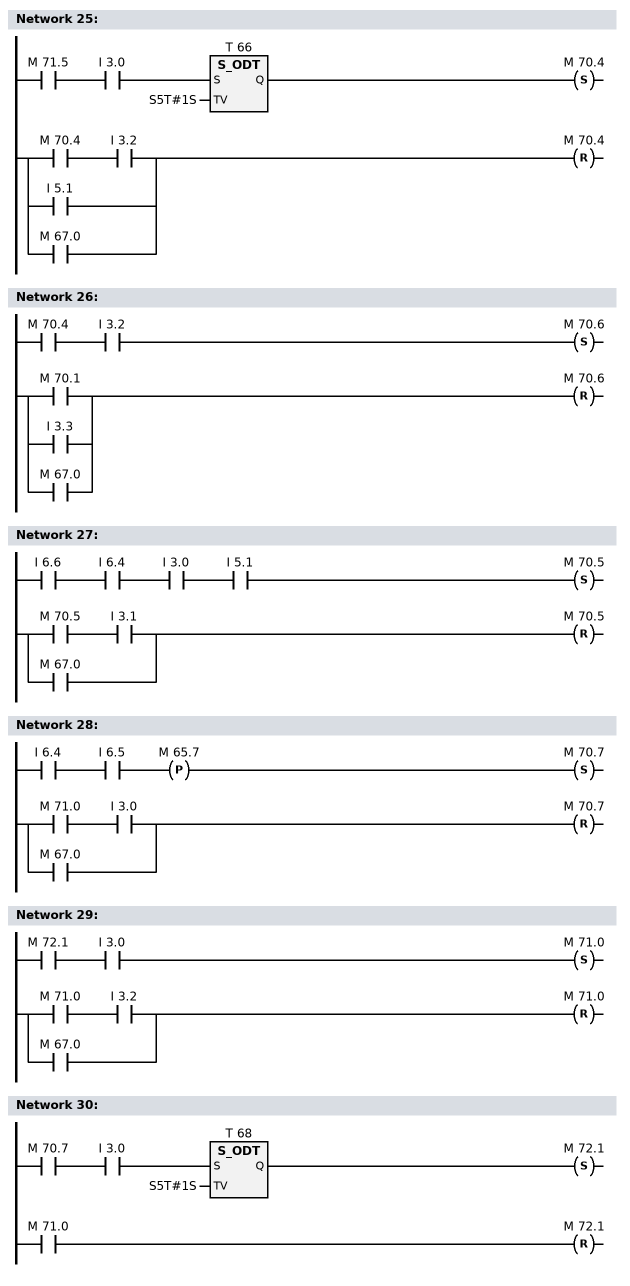
NETWORK
TITLE =
      A(;
      A     M 71.5;
      A     I 3.0;
      L     S5T#1S;
      SD    T 66;
      NOP   0;
      NOP   0;
      NOP   0;
      A     T 66;
      );
      S     M 70.4;
      A(;
      A     M 70.4;
      A     I 3.2;
      O     I 5.1;
      O     M 67.0;
      );
      R     M 70.4;
      NOP   0;
NETWORK
TITLE =
      A     M 70.4;
      A     I 3.2;
      S     M 70.6;
      A(;
      O     M 70.1;
      O     I 3.3;
      O     M 67.0;
      );
      R     M 70.6;
      NOP   0;
NETWORK
TITLE =
      A     I 6.6;
      A     I 6.4;
      A     I 3.0;
      A     I 5.1;
      S     M 70.5;
      A(;
      A     M 70.5;
      A     I 3.1;
      O     M 67.0;
      );
      R     M 70.5;
      NOP   0;
NETWORK
TITLE =
      A     I 6.4;
      A     I 6.5;
      FP    M 65.7;
      S     M 70.7;
      A(;
      A     M 71.0;
      A     I 3.0;
      O     M 67.0;
      );
      R     M 70.7;
      NOP   0;
NETWORK
TITLE =
      A     M 72.1;
      A     I 3.0;
      S     M 71.0;
      A(;
      A     M 71.0;
      A     I 3.2;
      O     M 67.0;
      );
      R     M 71.0;
      NOP   0;
NETWORK
TITLE =
      A(;
      A     M 70.7;
      A     I 3.0;
      L     S5T#1S;
      SD    T 68;
      NOP   0;
      NOP   0;
      NOP   0;
      A     T 68;
      );
      S     M 72.1;
      A     M 71.0;
      R     M 72.1;
      NOP   0;
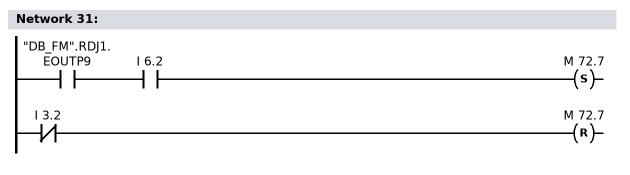
NETWORK
TITLE =
      A     "DB_FM".RDJ1.EOUTP9;
      A     I 6.2;
      S     M 72.7;
      AN    I 3.2;
      R     M 72.7;
      NOP   0;
END_FUNCTION

FUNCTION FC 115 : VOID
VERSION : 0.1
BEGIN
// (block stored without names or comments; labels and parameter names are numbered)
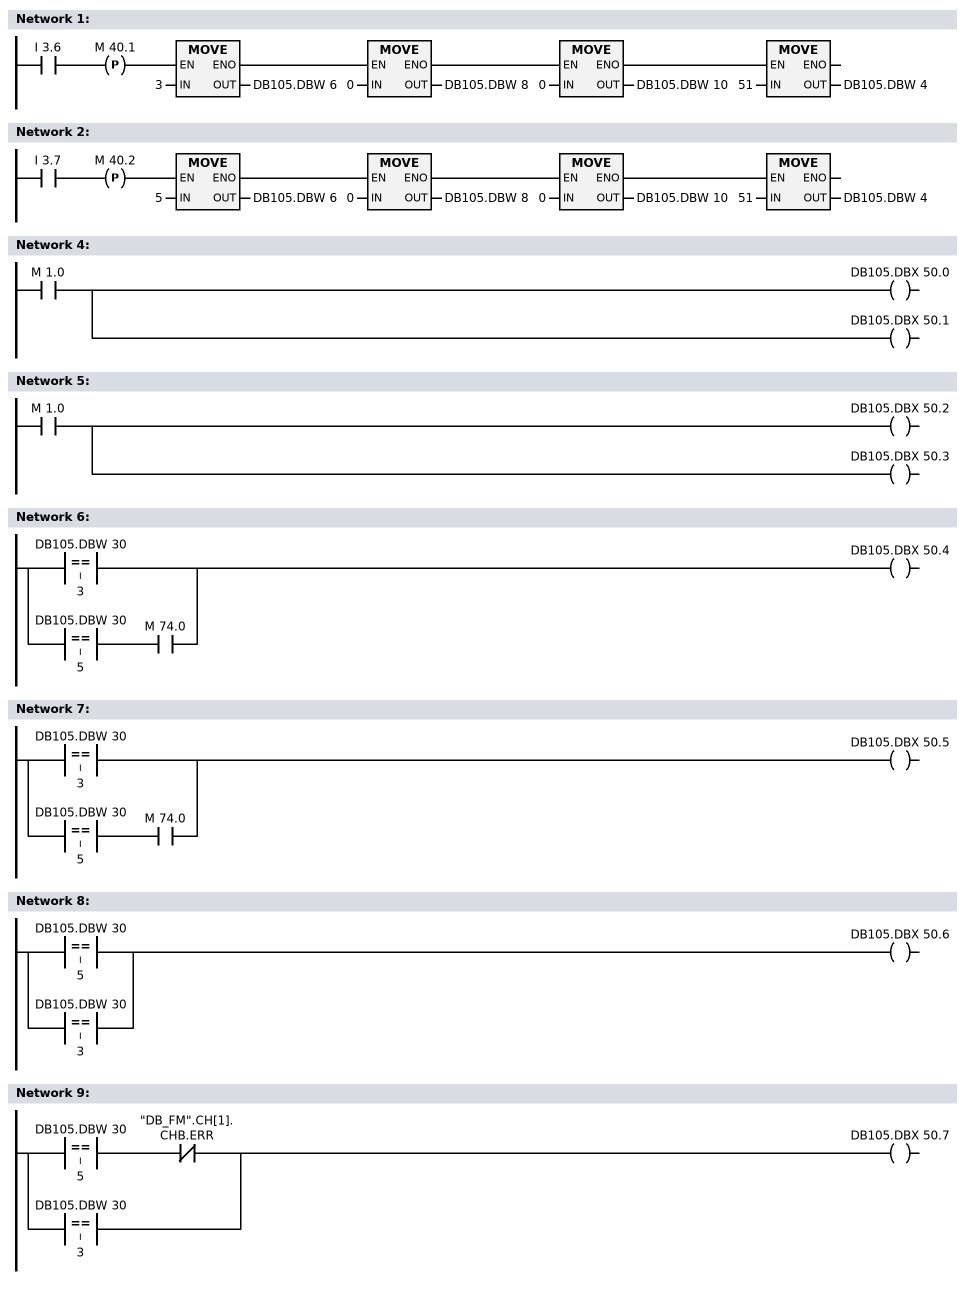
NETWORK
TITLE =
      A(;
      A(;
      A(;
      A     I 3.6;
      FP    M 40.1;
      JNB   M001;
      L     3;
      T     DB105.DBW 6;
      SET;
      SAVE;
      CLR;
M001: A     BR;
      );
      JNB   M002;
      L     0;
      T     DB105.DBW 8;
      SET;
      SAVE;
      CLR;
M002: A     BR;
      );
      JNB   M003;
      L     0;
      T     DB105.DBW 10;
      SET;
      SAVE;
      CLR;
M003: A     BR;
      );
      JNB   M004;
      L     51;
      T     DB105.DBW 4;
M004: NOP   0;
NETWORK
TITLE =
      A(;
      A(;
      A(;
      A     I 3.7;
      FP    M 40.2;
      JNB   M005;
      L     5;
      T     DB105.DBW 6;
      SET;
      SAVE;
      CLR;
M005: A     BR;
      );
      JNB   M006;
      L     0;
      T     DB105.DBW 8;
      SET;
      SAVE;
      CLR;
M006: A     BR;
      );
      JNB   M007;
      L     0;
      T     DB105.DBW 10;
      SET;
      SAVE;
      CLR;
M007: A     BR;
      );
      JNB   M008;
      L     51;
      T     DB105.DBW 4;
M008: NOP   0;
NETWORK
TITLE =
NETWORK
TITLE =
      A     M 1.0;
      =     DB105.DBX 50.0;
      =     DB105.DBX 50.1;
NETWORK
TITLE =
      A     M 1.0;
      =     DB105.DBX 50.2;
      =     DB105.DBX 50.3;
NETWORK
TITLE =
      O(;
      L     DB105.DBW 30;
      L     3;
      ==I;
      );
      O;
      A(;
      L     DB105.DBW 30;
      L     5;
      ==I;
      );
      A     M 74.0;
      =     DB105.DBX 50.4;
NETWORK
TITLE =
      O(;
      L     DB105.DBW 30;
      L     3;
      ==I;
      );
      O;
      A(;
      L     DB105.DBW 30;
      L     5;
      ==I;
      );
      A     M 74.0;
      =     DB105.DBX 50.5;
NETWORK
TITLE =
      O(;
      L     DB105.DBW 30;
      L     5;
      ==I;
      );
      O(;
      L     DB105.DBW 30;
      L     3;
      ==I;
      );
      =     DB105.DBX 50.6;
NETWORK
TITLE =
      A(;
      L     DB105.DBW 30;
      L     5;
      ==I;
      );
      AN    "DB_FM".CH[1].CHB.ERR;
      O(;
      L     DB105.DBW 30;
      L     3;
      ==I;
      );
      =     DB105.DBX 50.7;
END_FUNCTION

FUNCTION FC 118 : VOID
VERSION : 0.1
BEGIN
// (block stored without names or comments; labels and parameter names are numbered)
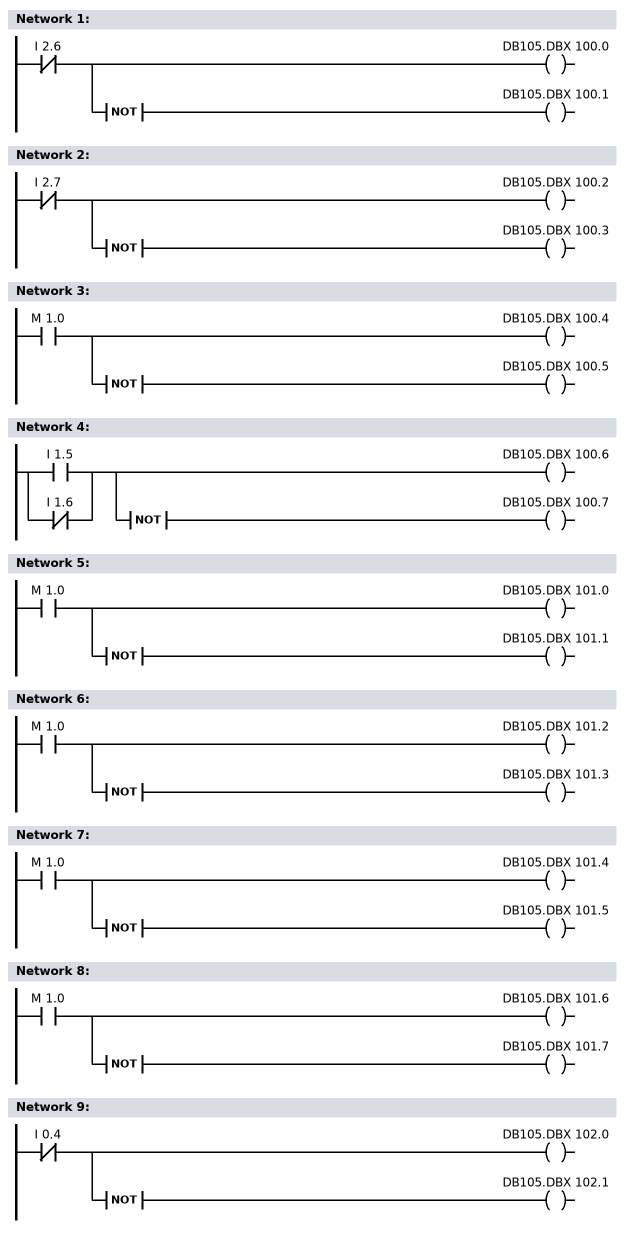
NETWORK
TITLE =
      AN    I 2.6;
      =     L 22.0;
      A     L 22.0;
      BLD   102;
      =     DB105.DBX 100.0;
      A     L 22.0;
      NOT;
      =     DB105.DBX 100.1;
NETWORK
TITLE =
      AN    I 2.7;
      =     L 22.0;
      A     L 22.0;
      BLD   102;
      =     DB105.DBX 100.2;
      A     L 22.0;
      NOT;
      =     DB105.DBX 100.3;
NETWORK
TITLE =
      A     M 1.0;
      =     L 22.0;
      A     L 22.0;
      BLD   102;
      =     DB105.DBX 100.4;
      A     L 22.0;
      NOT;
      =     DB105.DBX 100.5;
NETWORK
TITLE =
      O     I 1.5;
      ON    I 1.6;
      =     L 22.0;
      A     L 22.0;
      BLD   102;
      =     DB105.DBX 100.6;
      A     L 22.0;
      NOT;
      =     DB105.DBX 100.7;
NETWORK
TITLE =
      A     M 1.0;
      =     L 22.0;
      A     L 22.0;
      BLD   102;
      =     DB105.DBX 101.0;
      A     L 22.0;
      NOT;
      =     DB105.DBX 101.1;
NETWORK
TITLE =
      A     M 1.0;
      =     L 22.0;
      A     L 22.0;
      BLD   102;
      =     DB105.DBX 101.2;
      A     L 22.0;
      NOT;
      =     DB105.DBX 101.3;
NETWORK
TITLE =
      A     M 1.0;
      =     L 22.0;
      A     L 22.0;
      BLD   102;
      =     DB105.DBX 101.4;
      A     L 22.0;
      NOT;
      =     DB105.DBX 101.5;
NETWORK
TITLE =
      A     M 1.0;
      =     L 22.0;
      A     L 22.0;
      BLD   102;
      =     DB105.DBX 101.6;
      A     L 22.0;
      NOT;
      =     DB105.DBX 101.7;
NETWORK
TITLE =
      AN    I 0.4;
      =     L 22.0;
      A     L 22.0;
      BLD   102;
      =     DB105.DBX 102.0;
      A     L 22.0;
      NOT;
      =     DB105.DBX 102.1;
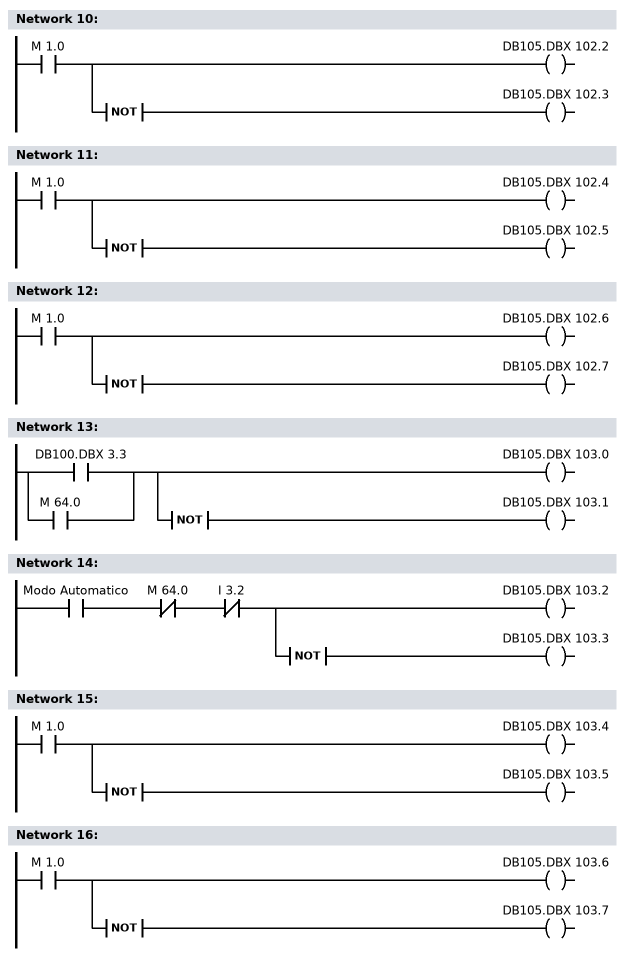
NETWORK
TITLE =
      A     M 1.0;
      =     L 22.0;
      A     L 22.0;
      BLD   102;
      =     DB105.DBX 102.2;
      A     L 22.0;
      NOT;
      =     DB105.DBX 102.3;
NETWORK
TITLE =
      A     M 1.0;
      =     L 22.0;
      A     L 22.0;
      BLD   102;
      =     DB105.DBX 102.4;
      A     L 22.0;
      NOT;
      =     DB105.DBX 102.5;
NETWORK
TITLE =
      A     M 1.0;
      =     L 22.0;
      A     L 22.0;
      BLD   102;
      =     DB105.DBX 102.6;
      A     L 22.0;
      NOT;
      =     DB105.DBX 102.7;
NETWORK
TITLE =
      O     DB100.DBX 3.3;
      O     M 64.0;
      =     L 22.0;
      A     L 22.0;
      BLD   102;
      =     DB105.DBX 103.0;
      A     L 22.0;
      NOT;
      =     DB105.DBX 103.1;
NETWORK
TITLE =
      A     "Modo Automatico";
      AN    M 64.0;
      AN    I 3.2;
      =     L 22.0;
      A     L 22.0;
      BLD   102;
      =     DB105.DBX 103.2;
      A     L 22.0;
      NOT;
      =     DB105.DBX 103.3;
NETWORK
TITLE =
      A     M 1.0;
      =     L 22.0;
      A     L 22.0;
      BLD   102;
      =     DB105.DBX 103.4;
      A     L 22.0;
      NOT;
      =     DB105.DBX 103.5;
NETWORK
TITLE =
      A     M 1.0;
      =     L 22.0;
      A     L 22.0;
      BLD   102;
      =     DB105.DBX 103.6;
      A     L 22.0;
      NOT;
      =     DB105.DBX 103.7;
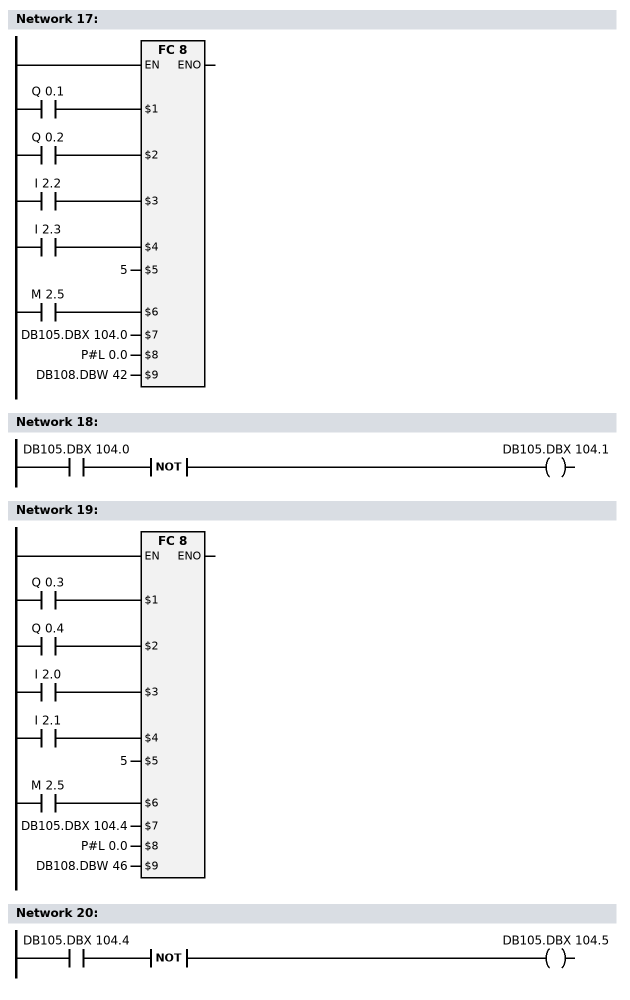
NETWORK
TITLE =
      A     Q 0.1;
      =     L 22.0;
      BLD   103;
      A     Q 0.2;
      =     L 22.1;
      BLD   103;
      A     I 2.2;
      =     L 22.2;
      BLD   103;
      A     I 2.3;
      =     L 22.3;
      BLD   103;
      A     M 2.5;
      =     L 22.4;
      BLD   103;
      CALL  FC 8 (
           $1                       := L 22.0,
           $2                       := L 22.1,
           $3                       := L 22.2,
           $4                       := L 22.3,
           $5                       := 5,
           $6                       := L 22.4,
           $7                       := DB105.DBX 104.0,
           $8                       := P#L 0.0,
           $9                       := DB108.DBW 42);
      NOP   0;
NETWORK
TITLE =
      A     DB105.DBX 104.0;
      NOT;
      =     DB105.DBX 104.1;
NETWORK
TITLE =
      A     Q 0.3;
      =     L 22.0;
      BLD   103;
      A     Q 0.4;
      =     L 22.1;
      BLD   103;
      A     I 2.0;
      =     L 22.2;
      BLD   103;
      A     I 2.1;
      =     L 22.3;
      BLD   103;
      A     M 2.5;
      =     L 22.4;
      BLD   103;
      CALL  FC 8 (
           $1                       := L 22.0,
           $2                       := L 22.1,
           $3                       := L 22.2,
           $4                       := L 22.3,
           $5                       := 5,
           $6                       := L 22.4,
           $7                       := DB105.DBX 104.4,
           $8                       := P#L 0.0,
           $9                       := DB108.DBW 46);
      NOP   0;
NETWORK
TITLE =
      A     DB105.DBX 104.4;
      NOT;
      =     DB105.DBX 104.5;
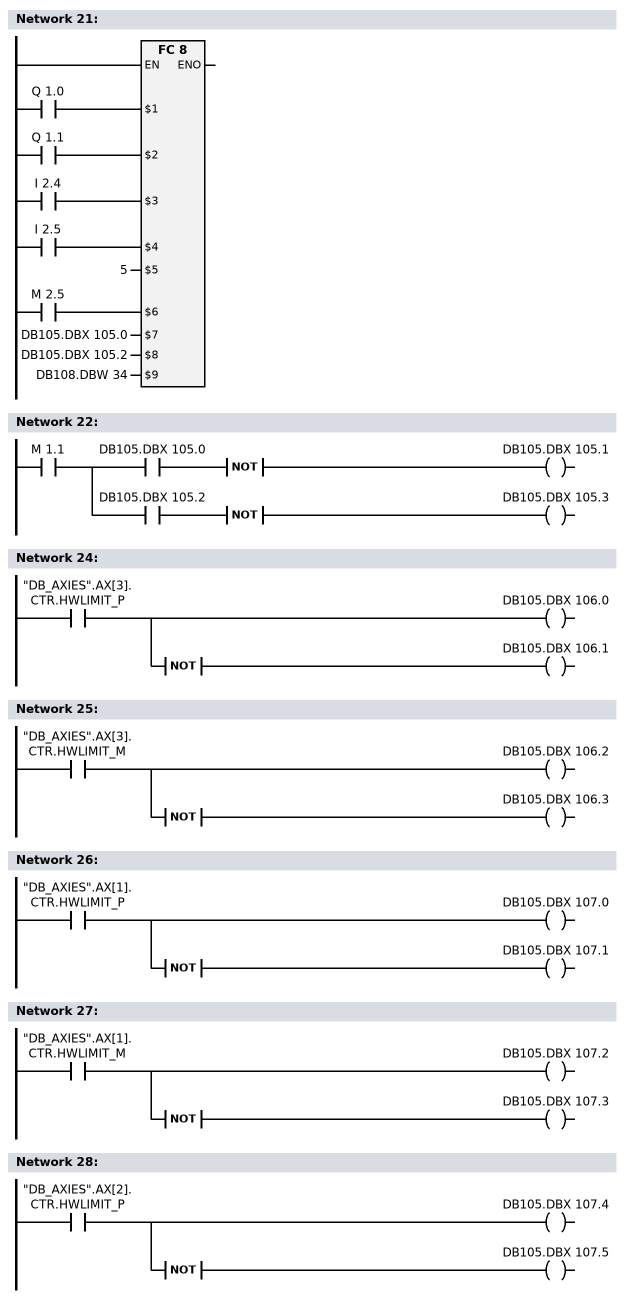
NETWORK
TITLE =
      A     Q 1.0;
      =     L 22.0;
      BLD   103;
      A     Q 1.1;
      =     L 22.1;
      BLD   103;
      A     I 2.4;
      =     L 22.2;
      BLD   103;
      A     I 2.5;
      =     L 22.3;
      BLD   103;
      A     M 2.5;
      =     L 22.4;
      BLD   103;
      CALL  FC 8 (
           $1                       := L 22.0,
           $2                       := L 22.1,
           $3                       := L 22.2,
           $4                       := L 22.3,
           $5                       := 5,
           $6                       := L 22.4,
           $7                       := DB105.DBX 105.0,
           $8                       := DB105.DBX 105.2,
           $9                       := DB108.DBW 34);
      NOP   0;
NETWORK
TITLE =
      A     M 1.1;
      =     L 22.0;
      A     L 22.0;
      A     DB105.DBX 105.0;
      NOT;
      =     DB105.DBX 105.1;
      A     L 22.0;
      A     DB105.DBX 105.2;
      NOT;
      =     DB105.DBX 105.3;
NETWORK
TITLE =
NETWORK
TITLE =
      A     "DB_AXIES".AX[3].CTR.HWLIMIT_P;
      =     L 22.0;
      A     L 22.0;
      BLD   102;
      =     DB105.DBX 106.0;
      A     L 22.0;
      NOT;
      =     DB105.DBX 106.1;
NETWORK
TITLE =
      A     "DB_AXIES".AX[3].CTR.HWLIMIT_M;
      =     L 22.0;
      A     L 22.0;
      BLD   102;
      =     DB105.DBX 106.2;
      A     L 22.0;
      NOT;
      =     DB105.DBX 106.3;
NETWORK
TITLE =
      A     "DB_AXIES".AX[1].CTR.HWLIMIT_P;
      =     L 22.0;
      A     L 22.0;
      BLD   102;
      =     DB105.DBX 107.0;
      A     L 22.0;
      NOT;
      =     DB105.DBX 107.1;
NETWORK
TITLE =
      A     "DB_AXIES".AX[1].CTR.HWLIMIT_M;
      =     L 22.0;
      A     L 22.0;
      BLD   102;
      =     DB105.DBX 107.2;
      A     L 22.0;
      NOT;
      =     DB105.DBX 107.3;
NETWORK
TITLE =
      A     "DB_AXIES".AX[2].CTR.HWLIMIT_P;
      =     L 22.0;
      A     L 22.0;
      BLD   102;
      =     DB105.DBX 107.4;
      A     L 22.0;
      NOT;
      =     DB105.DBX 107.5;
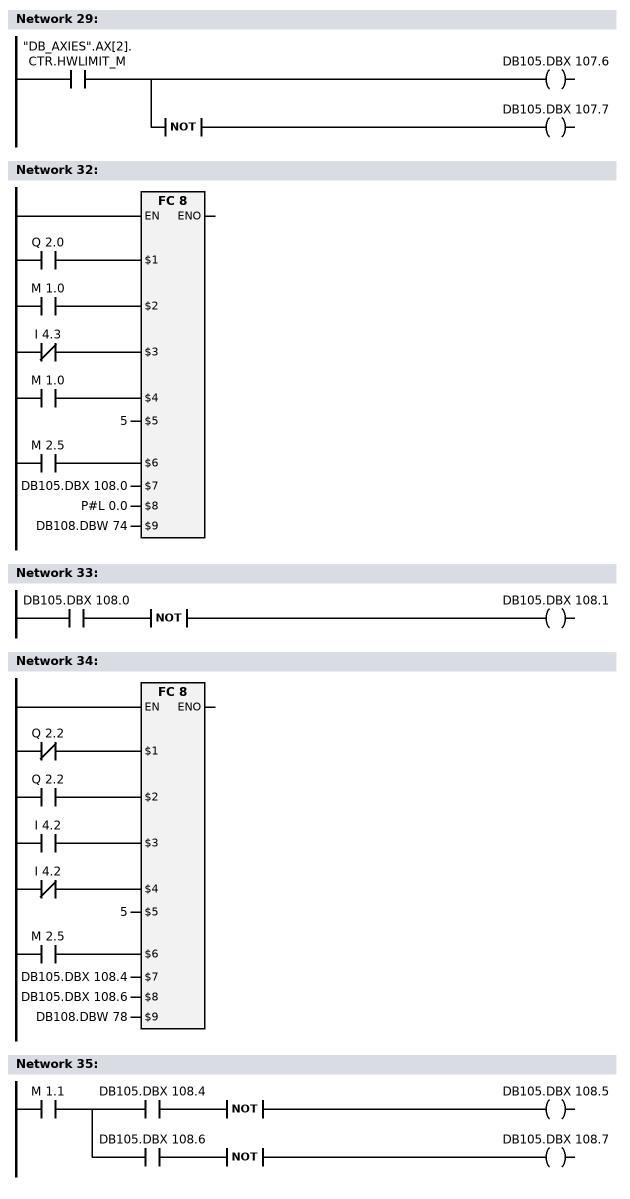
NETWORK
TITLE =
      A     "DB_AXIES".AX[2].CTR.HWLIMIT_M;
      =     L 22.0;
      A     L 22.0;
      BLD   102;
      =     DB105.DBX 107.6;
      A     L 22.0;
      NOT;
      =     DB105.DBX 107.7;
NETWORK
TITLE =
NETWORK
TITLE =
NETWORK
TITLE =
      A     Q 2.0;
      =     L 22.0;
      BLD   103;
      A     M 1.0;
      =     L 22.1;
      BLD   103;
      AN    I 4.3;
      =     L 22.2;
      BLD   103;
      A     M 1.0;
      =     L 22.3;
      BLD   103;
      A     M 2.5;
      =     L 22.4;
      BLD   103;
      CALL  FC 8 (
           $1                       := L 22.0,
           $2                       := L 22.1,
           $3                       := L 22.2,
           $4                       := L 22.3,
           $5                       := 5,
           $6                       := L 22.4,
           $7                       := DB105.DBX 108.0,
           $8                       := P#L 0.0,
           $9                       := DB108.DBW 74);
      NOP   0;
NETWORK
TITLE =
      A     DB105.DBX 108.0;
      NOT;
      =     DB105.DBX 108.1;
NETWORK
TITLE =
      AN    Q 2.2;
      =     L 22.0;
      BLD   103;
      A     Q 2.2;
      =     L 22.1;
      BLD   103;
      A     I 4.2;
      =     L 22.2;
      BLD   103;
      AN    I 4.2;
      =     L 22.3;
      BLD   103;
      A     M 2.5;
      =     L 22.4;
      BLD   103;
      CALL  FC 8 (
           $1                       := L 22.0,
           $2                       := L 22.1,
           $3                       := L 22.2,
           $4                       := L 22.3,
           $5                       := 5,
           $6                       := L 22.4,
           $7                       := DB105.DBX 108.4,
           $8                       := DB105.DBX 108.6,
           $9                       := DB108.DBW 78);
      NOP   0;
NETWORK
TITLE =
      A     M 1.1;
      =     L 22.0;
      A     L 22.0;
      A     DB105.DBX 108.4;
      NOT;
      =     DB105.DBX 108.5;
      A     L 22.0;
      A     DB105.DBX 108.6;
      NOT;
      =     DB105.DBX 108.7;
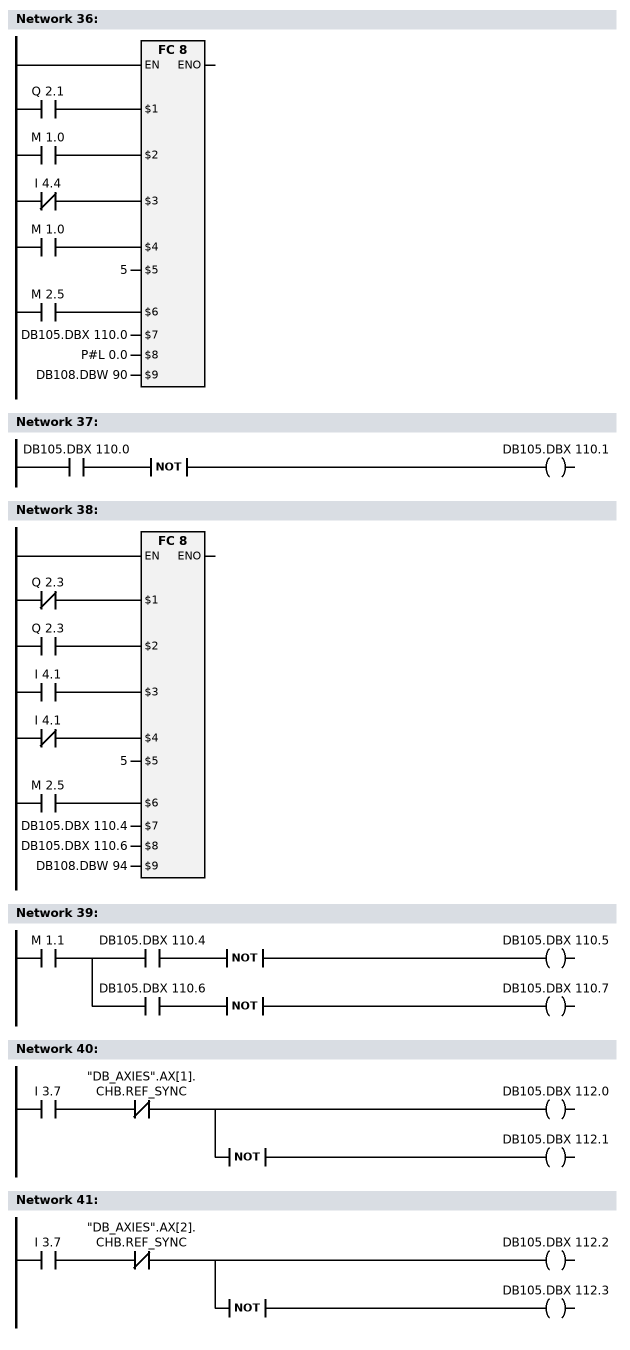
NETWORK
TITLE =
      A     Q 2.1;
      =     L 22.0;
      BLD   103;
      A     M 1.0;
      =     L 22.1;
      BLD   103;
      AN    I 4.4;
      =     L 22.2;
      BLD   103;
      A     M 1.0;
      =     L 22.3;
      BLD   103;
      A     M 2.5;
      =     L 22.4;
      BLD   103;
      CALL  FC 8 (
           $1                       := L 22.0,
           $2                       := L 22.1,
           $3                       := L 22.2,
           $4                       := L 22.3,
           $5                       := 5,
           $6                       := L 22.4,
           $7                       := DB105.DBX 110.0,
           $8                       := P#L 0.0,
           $9                       := DB108.DBW 90);
      NOP   0;
NETWORK
TITLE =
      A     DB105.DBX 110.0;
      NOT;
      =     DB105.DBX 110.1;
NETWORK
TITLE =
      AN    Q 2.3;
      =     L 22.0;
      BLD   103;
      A     Q 2.3;
      =     L 22.1;
      BLD   103;
      A     I 4.1;
      =     L 22.2;
      BLD   103;
      AN    I 4.1;
      =     L 22.3;
      BLD   103;
      A     M 2.5;
      =     L 22.4;
      BLD   103;
      CALL  FC 8 (
           $1                       := L 22.0,
           $2                       := L 22.1,
           $3                       := L 22.2,
           $4                       := L 22.3,
           $5                       := 5,
           $6                       := L 22.4,
           $7                       := DB105.DBX 110.4,
           $8                       := DB105.DBX 110.6,
           $9                       := DB108.DBW 94);
      NOP   0;
NETWORK
TITLE =
      A     M 1.1;
      =     L 22.0;
      A     L 22.0;
      A     DB105.DBX 110.4;
      NOT;
      =     DB105.DBX 110.5;
      A     L 22.0;
      A     DB105.DBX 110.6;
      NOT;
      =     DB105.DBX 110.7;
NETWORK
TITLE =
      A     I 3.7;
      AN    "DB_AXIES".AX[1].CHB.REF_SYNC;
      =     L 22.0;
      A     L 22.0;
      BLD   102;
      =     DB105.DBX 112.0;
      A     L 22.0;
      NOT;
      =     DB105.DBX 112.1;
NETWORK
TITLE =
      A     I 3.7;
      AN    "DB_AXIES".AX[2].CHB.REF_SYNC;
      =     L 22.0;
      A     L 22.0;
      BLD   102;
      =     DB105.DBX 112.2;
      A     L 22.0;
      NOT;
      =     DB105.DBX 112.3;
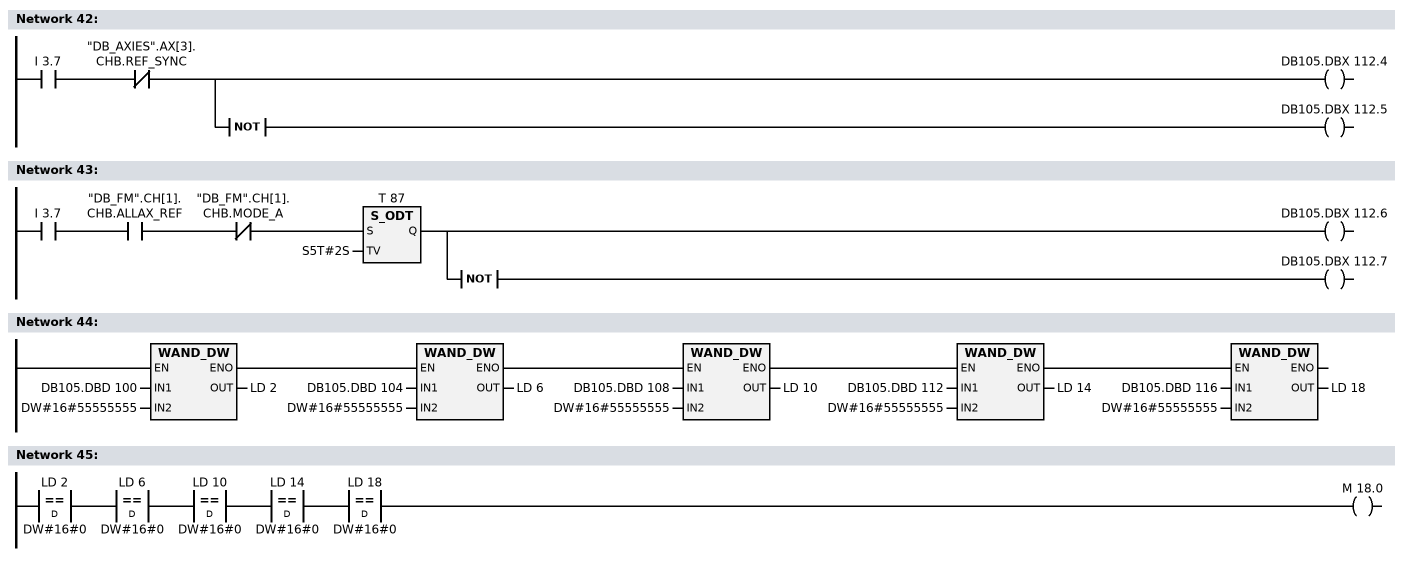
NETWORK
TITLE =
      A     I 3.7;
      AN    "DB_AXIES".AX[3].CHB.REF_SYNC;
      =     L 22.0;
      A     L 22.0;
      BLD   102;
      =     DB105.DBX 112.4;
      A     L 22.0;
      NOT;
      =     DB105.DBX 112.5;
NETWORK
TITLE =
      A     I 3.7;
      A     "DB_FM".CH[1].CHB.ALLAX_REF;
      AN    "DB_FM".CH[1].CHB.MODE_A;
      L     S5T#2S;
      SD    T 87;
      NOP   0;
      NOP   0;
      NOP   0;
      A     T 87;
      =     L 22.0;
      A     L 22.0;
      BLD   102;
      =     DB105.DBX 112.6;
      A     L 22.0;
      NOT;
      =     DB105.DBX 112.7;
NETWORK
TITLE =
      A(;
      A(;
      A(;
      A(;
      L     DB105.DBD 100;
      L     DW#16#55555555;
      AD;
      T     LD 2;
      SET;
      SAVE;
      CLR;
      A     BR;
      );
      JNB   M001;
      L     DB105.DBD 104;
      L     DW#16#55555555;
      AD;
      T     LD 6;
      SET;
      SAVE;
      CLR;
M001: A     BR;
      );
      JNB   M002;
      L     DB105.DBD 108;
      L     DW#16#55555555;
      AD;
      T     LD 10;
      SET;
      SAVE;
      CLR;
M002: A     BR;
      );
      JNB   M003;
      L     DB105.DBD 112;
      L     DW#16#55555555;
      AD;
      T     LD 14;
      SET;
      SAVE;
      CLR;
M003: A     BR;
      );
      JNB   M004;
      L     DB105.DBD 116;
      L     DW#16#55555555;
      AD;
      T     LD 18;
M004: NOP   0;
NETWORK
TITLE =
      A(;
      L     LD 2;
      L     DW#16#0;
      ==D;
      );
      A(;
      L     LD 6;
      L     DW#16#0;
      ==D;
      );
      A(;
      L     LD 10;
      L     DW#16#0;
      ==D;
      );
      A(;
      L     LD 14;
      L     DW#16#0;
      ==D;
      );
      A(;
      L     LD 18;
      L     DW#16#0;
      ==D;
      );
      =     M 18.0;
END_FUNCTION

FUNCTION FC 119 : VOID
VERSION : 0.1
BEGIN
// (block stored without names or comments; labels and parameter names are numbered)
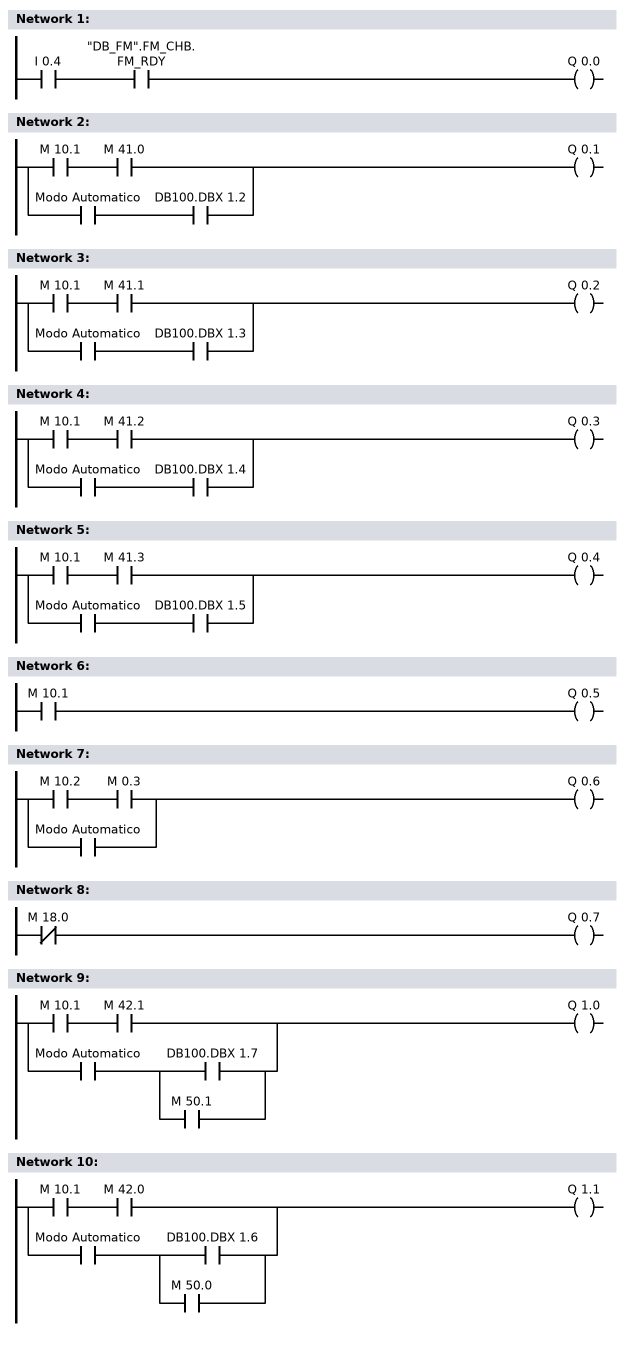
NETWORK
TITLE =
      A     I 0.4;
      A     "DB_FM".FM_CHB.FM_RDY;
      =     Q 0.0;
NETWORK
TITLE =
      A     M 10.1;
      A     M 41.0;
      O;
      A     "Modo Automatico";
      A     DB100.DBX 1.2;
      =     Q 0.1;
NETWORK
TITLE =
      A     M 10.1;
      A     M 41.1;
      O;
      A     "Modo Automatico";
      A     DB100.DBX 1.3;
      =     Q 0.2;
NETWORK
TITLE =
      A     M 10.1;
      A     M 41.2;
      O;
      A     "Modo Automatico";
      A     DB100.DBX 1.4;
      =     Q 0.3;
NETWORK
TITLE =
      A     M 10.1;
      A     M 41.3;
      O;
      A     "Modo Automatico";
      A     DB100.DBX 1.5;
      =     Q 0.4;
NETWORK
TITLE =
      A     M 10.1;
      =     Q 0.5;
NETWORK
TITLE =
      A     M 10.2;
      A     M 0.3;
      O     "Modo Automatico";
      =     Q 0.6;
NETWORK
TITLE =
      AN    M 18.0;
      =     Q 0.7;
NETWORK
TITLE =
      A     M 10.1;
      A     M 42.1;
      O;
      A     "Modo Automatico";
      A(;
      O     DB100.DBX 1.7;
      O     M 50.1;
      );
      =     Q 1.0;
NETWORK
TITLE =
      A     M 10.1;
      A     M 42.0;
      O;
      A     "Modo Automatico";
      A(;
      O     DB100.DBX 1.6;
      O     M 50.0;
      );
      =     Q 1.1;
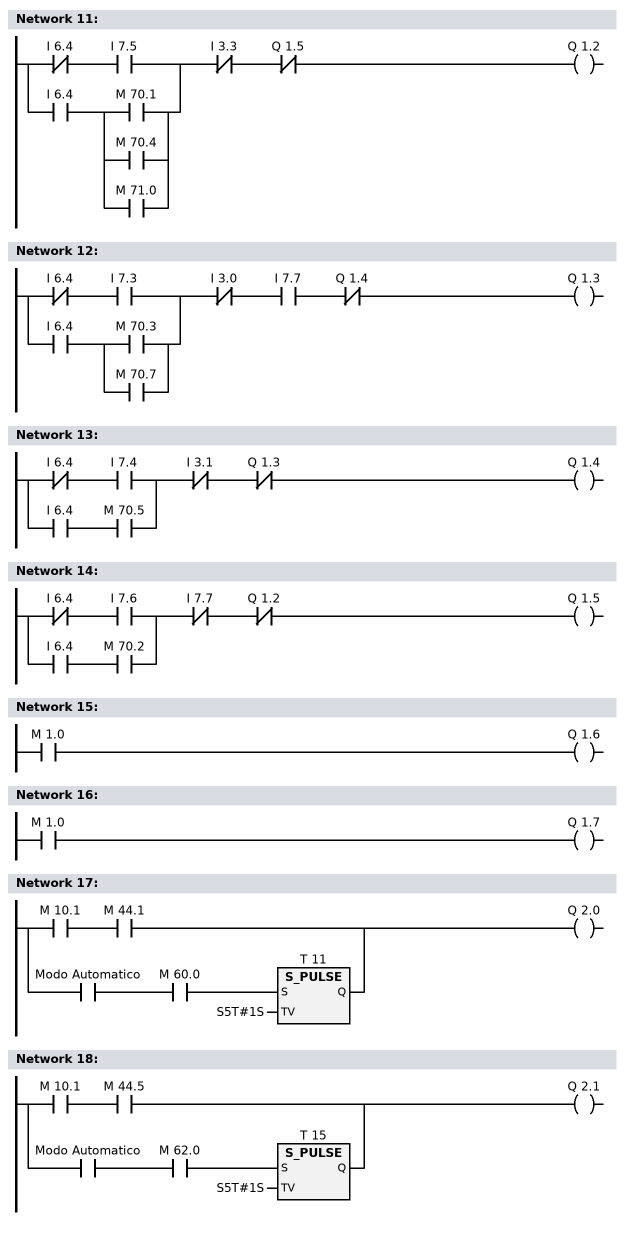
NETWORK
TITLE =
      A(;
      AN    I 6.4;
      A     I 7.5;
      O;
      A     I 6.4;
      A(;
      O     M 70.1;
      O     M 70.4;
      O     M 71.0;
      );
      );
      AN    I 3.3;
      AN    Q 1.5;
      =     Q 1.2;
NETWORK
TITLE =
      A(;
      AN    I 6.4;
      A     I 7.3;
      O;
      A     I 6.4;
      A(;
      O     M 70.3;
      O     M 70.7;
      );
      );
      AN    I 3.0;
      A     I 7.7;
      AN    Q 1.4;
      =     Q 1.3;
NETWORK
TITLE =
      A(;
      AN    I 6.4;
      A     I 7.4;
      O;
      A     I 6.4;
      A     M 70.5;
      );
      AN    I 3.1;
      AN    Q 1.3;
      =     Q 1.4;
NETWORK
TITLE =
      A(;
      AN    I 6.4;
      A     I 7.6;
      O;
      A     I 6.4;
      A     M 70.2;
      );
      AN    I 7.7;
      AN    Q 1.2;
      =     Q 1.5;
NETWORK
TITLE =
      A     M 1.0;
      =     Q 1.6;
NETWORK
TITLE =
      A     M 1.0;
      =     Q 1.7;
NETWORK
TITLE =
      A     M 10.1;
      A     M 44.1;
      O(;
      A     "Modo Automatico";
      A     M 60.0;
      L     S5T#1S;
      SP    T 11;
      NOP   0;
      NOP   0;
      NOP   0;
      A     T 11;
      );
      =     Q 2.0;
NETWORK
TITLE =
      A     M 10.1;
      A     M 44.5;
      O(;
      A     "Modo Automatico";
      A     M 62.0;
      L     S5T#1S;
      SP    T 15;
      NOP   0;
      NOP   0;
      NOP   0;
      A     T 15;
      );
      =     Q 2.1;
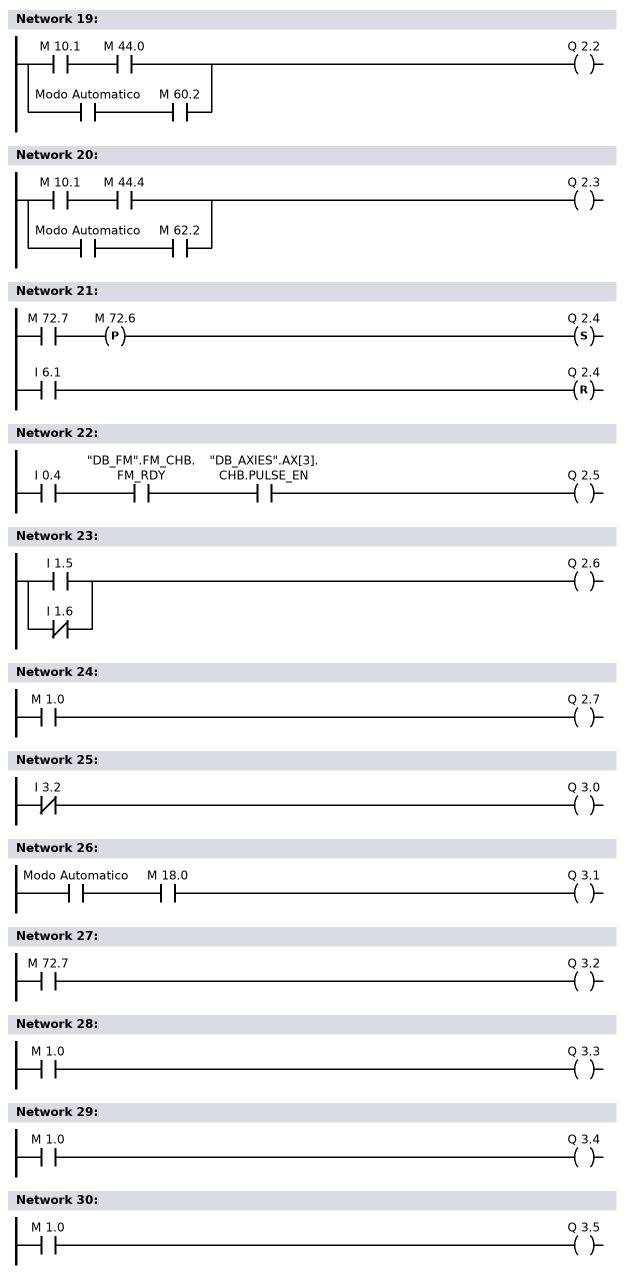
NETWORK
TITLE =
      A     M 10.1;
      A     M 44.0;
      O;
      A     "Modo Automatico";
      A     M 60.2;
      =     Q 2.2;
NETWORK
TITLE =
      A     M 10.1;
      A     M 44.4;
      O;
      A     "Modo Automatico";
      A     M 62.2;
      =     Q 2.3;
NETWORK
TITLE =
      A     M 72.7;
      FP    M 72.6;
      S     Q 2.4;
      A     I 6.1;
      R     Q 2.4;
      NOP   0;
NETWORK
TITLE =
      A     I 0.4;
      A     "DB_FM".FM_CHB.FM_RDY;
      A     "DB_AXIES".AX[3].CHB.PULSE_EN;
      =     Q 2.5;
NETWORK
TITLE =
      O     I 1.5;
      ON    I 1.6;
      =     Q 2.6;
NETWORK
TITLE =
      A     M 1.0;
      =     Q 2.7;
NETWORK
TITLE =
      AN    I 3.2;
      =     Q 3.0;
NETWORK
TITLE =
      A     "Modo Automatico";
      A     M 18.0;
      =     Q 3.1;
NETWORK
TITLE =
      A     M 72.7;
      =     Q 3.2;
NETWORK
TITLE =
      A     M 1.0;
      =     Q 3.3;
NETWORK
TITLE =
      A     M 1.0;
      =     Q 3.4;
NETWORK
TITLE =
      A     M 1.0;
      =     Q 3.5;
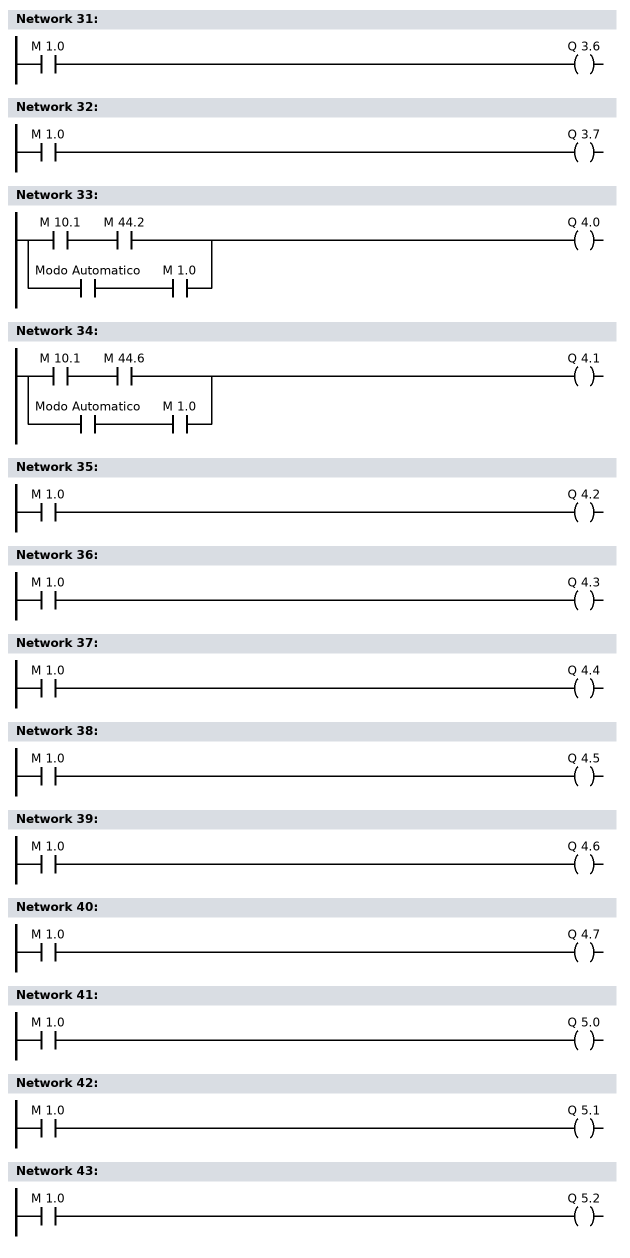
NETWORK
TITLE =
      A     M 1.0;
      =     Q 3.6;
NETWORK
TITLE =
      A     M 1.0;
      =     Q 3.7;
NETWORK
TITLE =
      A     M 10.1;
      A     M 44.2;
      O;
      A     "Modo Automatico";
      A     M 1.0;
      =     Q 4.0;
NETWORK
TITLE =
      A     M 10.1;
      A     M 44.6;
      O;
      A     "Modo Automatico";
      A     M 1.0;
      =     Q 4.1;
NETWORK
TITLE =
      A     M 1.0;
      =     Q 4.2;
NETWORK
TITLE =
      A     M 1.0;
      =     Q 4.3;
NETWORK
TITLE =
      A     M 1.0;
      =     Q 4.4;
NETWORK
TITLE =
      A     M 1.0;
      =     Q 4.5;
NETWORK
TITLE =
      A     M 1.0;
      =     Q 4.6;
NETWORK
TITLE =
      A     M 1.0;
      =     Q 4.7;
NETWORK
TITLE =
      A     M 1.0;
      =     Q 5.0;
NETWORK
TITLE =
      A     M 1.0;
      =     Q 5.1;
NETWORK
TITLE =
      A     M 1.0;
      =     Q 5.2;
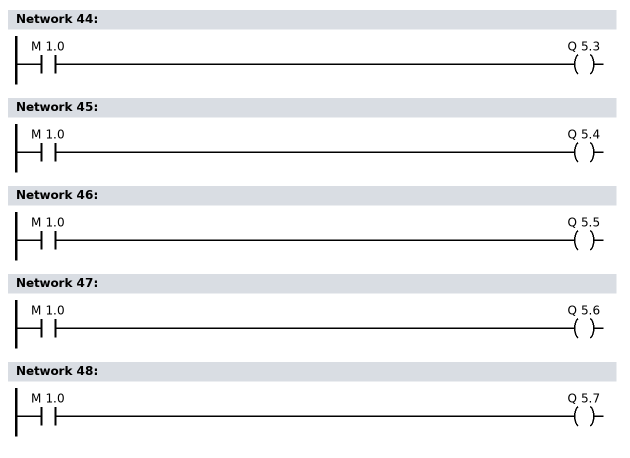
NETWORK
TITLE =
      A     M 1.0;
      =     Q 5.3;
NETWORK
TITLE =
      A     M 1.0;
      =     Q 5.4;
NETWORK
TITLE =
      A     M 1.0;
      =     Q 5.5;
NETWORK
TITLE =
      A     M 1.0;
      =     Q 5.6;
NETWORK
TITLE =
      A     M 1.0;
      =     Q 5.7;
END_FUNCTION

DATA_BLOCK DB 2
VERSION : 0.0
BEGIN
// 66 bytes; values not shown
END_DATA_BLOCK

// DB 7: know-how protected block, not included

DATA_BLOCK DB 15
AUTHOR : AuD_MCE8
FAMILY : FM357_2
NAME : BF_DB15
VERSION : 2.1
FB 6
BEGIN
END_DATA_BLOCK

// DB 16: know-how protected block, not included

// DB 17: know-how protected block, not included

// DB 19: know-how protected block, not included

// DB 20: know-how protected block, not included

DATA_BLOCK "DB_FM"	// DB 30
VERSION : 0.1
  STRUCT
   MOD_ADDR : INT ;	// Module address
   CH_NO : BYTE ;	// No. of channels
   AX_NO : BYTE ;	// No. of axes
   BF_ERR : WORD ;	// Basic function error
   WRJOB1 : BOOL ;	// Write request 1
   WRJOB2 : BOOL ;	// Write request 2
   BIT6_2 : BOOL ;	// Reserved
   BIT6_3 : BOOL ;	// Reserved
   BIT6_4 : BOOL ;	// Reserved
   BIT6_5 : BOOL ;	// Reserved
   BIT6_6 : BOOL ;	// Reserved
   BIT6_7 : BOOL ;	// Reserved
   ERR_WRJOB1 : BOOL ;	// Error in write request 1
   ERR_WRJOB2 : BOOL ;	// Error in write request 2
   BIT7_2 : BOOL ;	// Reserved
   BIT7_3 : BOOL ;	// Reserved
   BIT7_4 : BOOL ;	// Reserved
   BIT7_5 : BOOL ;	// Reserved
   BIT7_6 : BOOL ;	// Reserved
   BIT7_7 : BOOL ;	// Reserved
   RDJOB1 : BOOL ;	// Read request 1
   RDJOB2 : BOOL ;	// Read request 2
   BIT8_2 : BOOL ;	// Reserved
   BIT8_3 : BOOL ;	// Reserved
   BIT8_4 : BOOL ;	// Reserved
   BIT8_5 : BOOL ;	// Reserved
   BIT8_6 : BOOL ;	// Reserved
   BIT8_7 : BOOL ;	// Reserved
   ERR_RDJOB1 : BOOL ;	// Error in read request 1
   ERR_RDJOB2 : BOOL ;	// Error in read request 2
   BIT9_2 : BOOL ;	// Reserved
   BIT9_3 : BOOL ;	// Reserved
   BIT9_4 : BOOL ;	// Reserved
   BIT9_5 : BOOL ;	// Reserved
   BIT9_6 : BOOL ;	// Reserved
   BIT9_7 : BOOL ;	// Reserved
   CONNECT : BOOL ;	// Readiness to communicate
   RESTART : BOOL ;	// FM Restart
   STARTUP : BOOL ;	// FM Startup
   BIT10_3 : BOOL ;	// Reserved
   BIT10_4 : BOOL ;	// Reserved
   BIT10_5 : BOOL ;	// Reserved
   BIT10_6 : BOOL ;	// Reserved
   BIT10_7 : BOOL ;	// Reserved
   PRES_TEST : BOOL ;	// Start-up window: Request for TEST mode
   ACT_TEST : BOOL ;	// User: Enable TEST mode
   BIT11_2 : BOOL ;	// Reserved
   BIT11_3 : BOOL ;	// Reserved
   BIT11_4 : BOOL ;	// Reserved
   BIT11_5 : BOOL ;	// Reserved
   BIT11_6 : BOOL ;	// Reserved
   BIT11_7 : BOOL ;	// Reserved
   BYTE12_19 : ARRAY  [1 .. 8 ] OF BYTE ;	// Reserved
   FM_CTR : STRUCT 	// FM CONTROL SIGNALS
    BIT0_0 : BOOL ;	// Reserved
    EM_STOP : BOOL ;	// EMERGENCY STOP
    ACKN_EM_STOP : BOOL ;	// EMERGENCY STOP acknowledgement
    BIT0_3 : BOOL ;	// Reserved
    BIT0_4 : BOOL ;	// Reserved
    BIT0_5 : BOOL ;	// Reserved
    BIT0_6 : BOOL ;	// Reserved
    BIT0_7 : BOOL ;	// Reserved
    BIT1_0 : BOOL ;	// Reserved
    ACT_POS : BOOL ;	// Request actual values
    DIS_TOGO : BOOL ;	// Request distances to go
    BIT1_3 : BOOL ;	// Reserved
    BIT1_4 : BOOL ;	// Reserved
    BIT1_5 : BOOL ;	// Reserved
    BIT1_6 : BOOL ;	// Reserved
    BIT1_7 : BOOL ;	// Reserved
    CPU_VAR : WORD ;	// CPU variables(write)
    BYTE4_9 : ARRAY  [1 .. 6 ] OF BYTE ;	// Reserved
   END_STRUCT ;
   FM_CHB : STRUCT 	// FM CHECKBACK SIGNALS
    PROBE1 : BOOL ;	// Probe 1 actuated
    PROBE2 : BOOL ;	// Probe 2 actuated
    BIT0_2 : BOOL ;	// Reserved
    BIT0_3 : BOOL ;	// Reserved
    BIT0_4 : BOOL ;	// Reserved
    BIT0_5 : BOOL ;	// Reserved
    BIT0_6 : BOOL ;	// Reserved
    FM_RDY : BOOL ;	// FM ready
    FM_ERR : BOOL ;	// FM error is active
    EM_STOP : BOOL ;	// EMERGENCY STOP active
    BIT1_2 : BOOL ;	// Reserved
    BIT1_3 : BOOL ;	// Reserved
    BIT1_4 : BOOL ;	// Reserved
    BIT1_5 : BOOL ;	// Reserved
    BIT1_6 : BOOL ;	// Reserved
    BATT_ERR : BOOL ;	// FM battery fault
    SWCAM_M1 : BOOL ;	// Software cam MINUS 1
    SWCAM_M2 : BOOL ;	// Software cam MINUS 2
    SWCAM_M3 : BOOL ;	// Software cam MINUS 3
    SWCAM_M4 : BOOL ;	// Software cam MINUS 4
    SWCAM_M5 : BOOL ;	// Software cam MINUS 5
    SWCAM_M6 : BOOL ;	// Software cam MINUS 6
    SWCAM_M7 : BOOL ;	// Software cam MINUS 7
    SWCAM_M8 : BOOL ;	// Software cam MINUS 8
    SWCAM_P1 : BOOL ;	// Software cam PLUS 1
    SWCAM_P2 : BOOL ;	// Software cam PLUS 2
    SWCAM_P3 : BOOL ;	// Software cam PLUS 3
    SWCAM_P4 : BOOL ;	// Software cam PLUS 4
    SWCAM_P5 : BOOL ;	// Software cam PLUS 5
    SWCAM_P6 : BOOL ;	// Software cam PLUS 6
    SWCAM_P7 : BOOL ;	// Software cam PLUS 7
    SWCAM_P8 : BOOL ;	// Software cam PLUS 8
    CPU_VAR : WORD ;	// CPU variables (read)
    BYTE6_9 : ARRAY  [1 .. 4 ] OF BYTE ;	// Reserved
   END_STRUCT ;
   BYTE40_99 : ARRAY  [1 .. 60 ] OF BYTE ;	// Reserved
   CH : ARRAY  [1 .. 4 ] OF STRUCT 	// CHANNEL SIGNALS
    CTR : STRUCT 	// CHANNEL CONTROL SIGNALS
     MODE_A : BOOL ;	// Automatic mode
     MODE_MDI : BOOL ;	// MDI block mode (FM357-H)
     MODE_JOG : BOOL ;	// Jog mode
     BIT0_3 : BOOL ;	// Reserved
     BIT0_4 : BOOL ;	// Reserved
     BIT0_5 : BOOL ;	// Reserved
     BIT0_6 : BOOL ;	// Reserved
     BIT0_7 : BOOL ;	// Reserved
     TEACH_IN : BOOL ;	// Teach-In (FM357-H)
     REPOS : BOOL ;	// Repositioning (FM357-H)
     REF_POINT : BOOL ;	// Reference point approach
     BIT1_3 : BOOL ;	// Reserved
     BIT1_4 : BOOL ;	// Reserved
     BIT1_5 : BOOL ;	// Reserved
     BIT1_6 : BOOL ;	// Reserved
     BIT1_7 : BOOL ;	// Reserved
     INC1 : BOOL ;	// Increment size 1 increment
     INC10 : BOOL ;	// Increment size 10 increments
     INC100 : BOOL ;	// Increment size 100 increments
     INC1000 : BOOL ;	// Increment size 1000 increments
     INC10000 : BOOL ;	// Increment size 10000 increments
     INC_VAR : BOOL ;	// Increment variable (FM357-H)
     CONT_TRAV : BOOL ;	// Continuous traverse
     BIT2_7 : BOOL ;	// Reserved
     BIT3_0 : BOOL ;	// Reserved
     BIT3_1 : BOOL ;	// Reserved
     BIT3_2 : BOOL ;	// Reserved
     BIT3_3 : BOOL ;	// Reserved
     SGL_BL : BOOL ;	// Activate single block
     M1 : BOOL ;	// Activate M1
     DRUN_FD : BOOL ;	// Dry run feed (FM357-H)
     BIT3_7 : BOOL ;	// Reserved
     BIT4_0 : BOOL ;	// Reserved
     BIT4_1 : BOOL ;	// Reserved
     BIT4_2 : BOOL ;	// Reserved
     BIT4_3 : BOOL ;	// Reserved
     BIT4_4 : BOOL ;	// Reserved
     BIT4_5 : BOOL ;	// Reserved
     BIT4_6 : BOOL ;	// Reserved
     PROG_TEST : BOOL ;	// Activate program test (FM357-H)
     SKIP_BL : BOOL ;	// Activate skip block
     BIT5_1 : BOOL ;	// Reserved
     BIT5_2 : BOOL ;	// Reserved
     BIT5_3 : BOOL ;	// Reserved
     BIT5_4 : BOOL ;	// Reserved
     BIT5_5 : BOOL ;	// Reserved
     BIT5_6 : BOOL ;	// Reserved
     BIT5_7 : BOOL ;	// Reserved
     FD_OVERR : BYTE ;	// Path override
     FD_DISA : BOOL ;	// Activate feed disable
     RDIN_DISA : BOOL ;	// Read-in disable
     DELDIS_TOGO : BOOL ;	// Delete distance to go
     BIT7_3 : BOOL ;	// Reserved
     BIT7_4 : BOOL ;	// Reserved
     BIT7_5 : BOOL ;	// Reserved
     FD_OVERR_RTR : BOOL ;	// Path override rapid traverse operative
     FD_OVERR_FDR : BOOL ;	// Path override feedrate operative
     START_DISA : BOOL ;	// Activate start disable
     START : BOOL ;	// Start
     STOP_BL : BOOL ;	// Activate stop at block limit
     STOP : BOOL ;	// Stop
     BIT8_4 : BOOL ;	// Reserved
     BIT8_5 : BOOL ;	// Reserved
     BIT8_6 : BOOL ;	// Reserved
     RESET : BOOL ;	// Reset
     ACKN_AUXILF : BOOL ;	// Acknowledge aux. function
     BIT9_1 : BOOL ;	// Reserved
     BIT9_2 : BOOL ;	// Reserved
     BIT9_3 : BOOL ;	// Reserved
     BIT9_4 : BOOL ;	// Reserved
     BIT9_5 : BOOL ;	// Reserved
     BIT9_6 : BOOL ;	// Reserved
     BIT9_7 : BOOL ;	// Reserved
     BIT10_0 : BOOL ;	// Reserved
     BIT10_1 : BOOL ;	// Reserved
     BIT10_2 : BOOL ;	// Reserved
     BIT10_3 : BOOL ;	// Reserved
     BIT10_4 : BOOL ;	// Reserved
     BIT10_5 : BOOL ;	// Reserved
     BIT10_6 : BOOL ;	// Reserved
     START_ASUP : BOOL ;	// Start "Asynchronous subroutine"
     BYTE11 : BYTE ;	// Reserved
     WORD12 : WORD ;	// Reserved
     BIT14_0 : BOOL ;	// Reserved
     BIT14_1 : BOOL ;	// Reserved
     BIT14_2 : BOOL ;	// Reserved
     FD_STOP_GEOA1 : BOOL ;	// Feed stop geometry axis 1 (FM357-H)
     TR_DISA_GEOA1 : BOOL ;	// Traverse disable geometry axis 1 (FM357-H)
     RTR_OVERL_GEOA1 : BOOL ;	// Rapid traverse override geometry axis 1 (FM357-H)
     DIR_M_GEOA1 : BOOL ;	// MINUS direction geometry axis  1(FM357-H)
     DIR_P_GEOA1 : BOOL ;	// PLUS direction geometry axis 1 (FM357-H)
     BIT15_0 : BOOL ;	// Reserved
     BIT15_1 : BOOL ;	// Reserved
     BIT15_2 : BOOL ;	// Reserved
     FD_STOP_GEOA2 : BOOL ;	// Feed stop geometry axis 2 (FM357-H)
     TR_DISA_GEOA2 : BOOL ;	// Traverse disable geometry axis 2 (FM357-H)
     RTR_OVERL_GEOA2 : BOOL ;	// Rapid traverse override geometry axis 2 (FM357-H)
     DIR_M_GEOA2 : BOOL ;	// MINUS direction geometry axis 2(FM357-H)
     DIR_P_GEOA2 : BOOL ;	// PLUS direction geometry axis 2 (FM357-H)
     BIT16_0 : BOOL ;	// Reserved
     BIT16_1 : BOOL ;	// Reserved
     BIT16_2 : BOOL ;	// Reserved
     FD_STOP_GEOA3 : BOOL ;	// Feed stop geometry axis 3 (FM357-H)
     TR_DISA_GEOA3 : BOOL ;	// Traverse disable geometry axis 3 (FM357-H)
     RTR_OVERL_GEOA3 : BOOL ;	// Rapid traverse override geometry axis 3 (FM357-H)
     DIR_M_GEOA3 : BOOL ;	// MINUS direction geometry axis 3 (FM357-H)
     DIR_P_GEOA3 : BOOL ;	// PLUS direction geometry axis 3 (FM357-H)
     BIT17_0 : BOOL ;	// Reserved
     BIT17_1 : BOOL ;	// Reserved
     BIT17_2 : BOOL ;	// Reserved
     FD_STOP_ORIA1 : BOOL ;	// Feed stop orientation axis 1 (FM357-H)
     TR_DISA_ORIA1 : BOOL ;	// Traverse disable orientation axis 1 (FM357-H)
     RTR_OVERL_ORIA1 : BOOL ;	// Rapid traverse override orientation axis 1 (FM357-H)
     DIR_M_ORIA1 : BOOL ;	// MINUS direction orientation axis 1 (FM357-H)
     DIR_P_ORIA1 : BOOL ;	// PLUS direction orientation axis 1 (FM357-H)
     WORD18 : WORD ;	// Reserved
    END_STRUCT ;
    CHB : STRUCT 	// CHANNEL CHECKBACK SIGNALS
     MODE_A : BOOL ;	// Automatic mode active
     MODE_MDI : BOOL ;	// MDI block mode active (FM357-H)
     MODE_JOG : BOOL ;	// Jog mode active
     BIT0_3 : BOOL ;	// Reserved
     BIT0_4 : BOOL ;	// Reserved
     BIT0_5 : BOOL ;	// Reserved
     BIT0_6 : BOOL ;	// Reserved
     BIT0_7 : BOOL ;	// Reserved
     TEACH_IN : BOOL ;	// Teach-In active (FM357-H)
     REPOS : BOOL ;	// Repositioning active (FM357-H)
     REF_POINT : BOOL ;	// Reference point approach active
     BIT1_3 : BOOL ;	// Reserved
     BIT1_4 : BOOL ;	// Reserved
     BIT1_5 : BOOL ;	// Reserved
     BIT1_6 : BOOL ;	// Reserved
     BIT1_7 : BOOL ;	// Reserved
     INC1 : BOOL ;	// Increment size 1 increment active
     INC10 : BOOL ;	// Increment size 10 increments active
     INC100 : BOOL ;	// Increment size 100 increments active
     INC1000 : BOOL ;	// Increment size 1000 increments active
     INC10000 : BOOL ;	// Increment size 10000 increments active
     INC_VAR : BOOL ;	// Increment variable (FM357-H)
     CONT_TRAV : BOOL ;	// Continuous traverse active
     BIT2_7 : BOOL ;	// Reserved
     BIT3_0 : BOOL ;	// Reserved
     BIT3_1 : BOOL ;	// Reserved
     BIT3_2 : BOOL ;	// Reserved
     BIT3_3 : BOOL ;	// Reserved
     BIT3_4 : BOOL ;	// Reserved
     M0_M1 : BOOL ;	// M0 / M1 active
     BIT3_6 : BOOL ;	// Reserved
     BIT3_7 : BOOL ;	// Reserved
     BIT4_0 : BOOL ;	// Reserved
     BIT4_1 : BOOL ;	// Reserved
     BIT4_2 : BOOL ;	// Reserved
     BIT4_3 : BOOL ;	// Reserved
     BIT4_4 : BOOL ;	// Reserved
     M2_M30 : BOOL ;	// M2 / M30 active
     TRANSF : BOOL ;	// Transformation active (FM357-H)
     PROG_TEST : BOOL ;	// Program test active (FM357-H)
     PROG_RUN : BOOL ;	// Program running
     PROG_WAIT : BOOL ;	// Program waiting
     PROG_STOP : BOOL ;	// Program stopped
     PROG_INT : BOOL ;	// Program interrupted
     PROG_AB : BOOL ;	// Program aborted
     BIT5_5 : BOOL ;	// Reserved
     BIT5_6 : BOOL ;	// Reserved
     RESET : BOOL ;	// Channel reset acknowledgement
     BIT6_0 : BOOL ;	// Reserved
     BIT6_1 : BOOL ;	// Reserved
     ALLAX_REF : BOOL ;	// All axes referenced
     ALLAX_STOP : BOOL ;	// All axes stationary
     BIT6_4 : BOOL ;	// Reserved
     CH_RDY : BOOL ;	// Channel ready
     ERR : BOOL ;	// Channel error
     ERR_STOP : BOOL ;	// Channel error; program stopped
     CHANG_AUXILF : BOOL ;	// Aux. function modification
     BIT7_1 : BOOL ;	// Reserved
     BIT7_2 : BOOL ;	// Reserved
     BIT7_3 : BOOL ;	// Reserved
     BIT7_4 : BOOL ;	// Reserved
     BIT7_5 : BOOL ;	// Reserved
     BIT7_6 : BOOL ;	// Reserved
     BIT7_7 : BOOL ;	// Reserved
     ASUP_ACT : BOOL ;	// "Asynchronous subroutine" active
     ASUP_DONE : BOOL ;	// "Asynchronous subroutine" ended
     ASUP_ERR : BOOL ;	// "Asynchronous subroutine" error
     ASUP_STARTERR : BOOL ;	// "Asynchronous subroutine" start error
     BIT8_4 : BOOL ;	// Reserved
     BIT8_5 : BOOL ;	// Reserved
     BIT8_6 : BOOL ;	// Reserved
     BIT8_7 : BOOL ;	// Reserved
     BYTE9 : BYTE ;	// Reserved
     WORD10 : WORD ;	// Reserved
     WORD12 : WORD ;	// Reserved
     BIT14_0 : BOOL ;	// Reserved
     BIT14_1 : BOOL ;	// Reserved
     BIT14_2 : BOOL ;	// Reserved
     BIT14_3 : BOOL ;	// Reserved
     BIT14_4 : BOOL ;	// Reserved
     BIT14_5 : BOOL ;	// Reserved
     GO_M_GEOA1 : BOOL ;	// Traverse MINUS geometry axis 1 (FM357-H)
     GO_P_GEOA1 : BOOL ;	// Traverse PLUS geometry axis 1 (FM357-H)
     BIT15_0 : BOOL ;	// Reserved
     BIT15_1 : BOOL ;	// Reserved
     BIT15_2 : BOOL ;	// Reserved
     BIT15_3 : BOOL ;	// Reserved
     BIT15_4 : BOOL ;	// Reserved
     BIT15_5 : BOOL ;	// Reserved
     GO_M_GEOA2 : BOOL ;	// Traverse MINUS geometry axis 2 (FM357-H)
     GO_P_GEOA2 : BOOL ;	// Traverse PLUS geometry axis 2 (FM357-H)
     BIT16_0 : BOOL ;	// Reserved
     BIT16_1 : BOOL ;	// Reserved
     BIT16_2 : BOOL ;	// Reserved
     BIT16_3 : BOOL ;	// Reserved
     BIT16_4 : BOOL ;	// Reserved
     BIT16_5 : BOOL ;	// Reserved
     GO_M_GEOA3 : BOOL ;	// Traverse MINUS geometry axis 3 (FM357-H)
     GO_P_GEOA3 : BOOL ;	// Traverse PLUS geometry axis 3 (FM357-H)
     BIT17_0 : BOOL ;	// Reserved
     BIT17_1 : BOOL ;	// Reserved
     BIT17_2 : BOOL ;	// Reserved
     BIT17_3 : BOOL ;	// Reserved
     BIT17_4 : BOOL ;	// Reserved
     BIT17_5 : BOOL ;	// Reserved
     GO_M_ORIA1 : BOOL ;	// Traverse MINUS orientation axis 1 (FM357-H)
     GO_P_ORIA1 : BOOL ;	// Traverse PLUS orientation axis 1 (FM357-H)
     WORD18 : WORD ;	// Reserved
    END_STRUCT ;
    AUXILF : STRUCT 	// CHANNEL AUX. FUNCTIONS
     MF0 : BOOL ;	// M function 0
     MF1 : BOOL ;	// M function 1
     MF2 : BOOL ;	// M function 2
     MF3 : BOOL ;	// M function 3
     MF4 : BOOL ;	// M function 4
     MF5 : BOOL ;	// M function 5
     MF6 : BOOL ;	// M function 6
     MF7 : BOOL ;	// M function 7
     MF8 : BOOL ;	// M function 8
     MF9 : BOOL ;	// M function 9
     MF10 : BOOL ;	// M function 10
     MF11 : BOOL ;	// M function 11
     MF12 : BOOL ;	// M function 12
     MF13 : BOOL ;	// M function 13
     MF14 : BOOL ;	// M function 14
     MF15 : BOOL ;	// M function 15
     MF16 : BOOL ;	// M function 16
     MF17 : BOOL ;	// M function 17
     MF18 : BOOL ;	// M function 18
     MF19 : BOOL ;	// M function 19
     MF20 : BOOL ;	// M function 20
     MF21 : BOOL ;	// M function 21
     MF22 : BOOL ;	// M function 22
     MF23 : BOOL ;	// M function 23
     MF24 : BOOL ;	// M function 24
     MF25 : BOOL ;	// M function 25
     MF26 : BOOL ;	// M function 26
     MF27 : BOOL ;	// M function 27
     MF28 : BOOL ;	// M function 28
     MF29 : BOOL ;	// M function 29
     MF30 : BOOL ;	// M function 30
     MF31 : BOOL ;	// M function 31
     MF32 : BOOL ;	// M function 32
     MF33 : BOOL ;	// M function 33
     MF34 : BOOL ;	// M function 34
     MF35 : BOOL ;	// M function 35
     MF36 : BOOL ;	// M function 36
     MF37 : BOOL ;	// M function 37
     MF38 : BOOL ;	// M function 38
     MF39 : BOOL ;	// M function 39
     MF40 : BOOL ;	// M function 40
     MF41 : BOOL ;	// M function 41
     MF42 : BOOL ;	// M function 42
     MF43 : BOOL ;	// M function 43
     MF44 : BOOL ;	// M function 44
     MF45 : BOOL ;	// M function 45
     MF46 : BOOL ;	// M function 46
     MF47 : BOOL ;	// M function 47
     MF48 : BOOL ;	// M function 48
     MF49 : BOOL ;	// M function 49
     MF50 : BOOL ;	// M function 50
     MF51 : BOOL ;	// M function 51
     MF52 : BOOL ;	// M function 52
     MF53 : BOOL ;	// M function 53
     MF54 : BOOL ;	// M function 54
     MF55 : BOOL ;	// M function 55
     MF56 : BOOL ;	// M function 56
     MF57 : BOOL ;	// M function 57
     MF58 : BOOL ;	// M function 58
     MF59 : BOOL ;	// M function 59
     MF60 : BOOL ;	// M function 60
     MF61 : BOOL ;	// M function 61
     MF62 : BOOL ;	// M function 62
     MF63 : BOOL ;	// M function 63
     MF64 : BOOL ;	// M function 64
     MF65 : BOOL ;	// M function 65
     MF66 : BOOL ;	// M function 66
     MF67 : BOOL ;	// M function 67
     MF68 : BOOL ;	// M function 68
     MF69 : BOOL ;	// M function 69
     MF70 : BOOL ;	// M function 70
     MF71 : BOOL ;	// M function 71
     MF72 : BOOL ;	// M function 72
     MF73 : BOOL ;	// M function 73
     MF74 : BOOL ;	// M function 74
     MF75 : BOOL ;	// M function 75
     MF76 : BOOL ;	// M function 76
     MF77 : BOOL ;	// M function 77
     MF78 : BOOL ;	// M function 78
     MF79 : BOOL ;	// M function 79
     MF80 : BOOL ;	// M function 80
     MF81 : BOOL ;	// M function 81
     MF82 : BOOL ;	// M function 82
     MF83 : BOOL ;	// M function 83
     MF84 : BOOL ;	// M function 84
     MF85 : BOOL ;	// M function 85
     MF86 : BOOL ;	// M function 86
     MF87 : BOOL ;	// M function 87
     MF88 : BOOL ;	// M function 88
     MF89 : BOOL ;	// M function 89
     MF90 : BOOL ;	// M function 90
     MF91 : BOOL ;	// M function 91
     MF92 : BOOL ;	// M function 92
     MF93 : BOOL ;	// M function 93
     MF94 : BOOL ;	// M function 94
     MF95 : BOOL ;	// M function 95
     MF96 : BOOL ;	// M function 96
     MF97 : BOOL ;	// M function 97
     MF98 : BOOL ;	// M function 98
     MF99 : BOOL ;	// M function 99
     BIT12_4 : BOOL ;	// Reserved
     BIT12_5 : BOOL ;	// Reserved
     BIT12_6 : BOOL ;	// Reserved
     BIT12_7 : BOOL ;	// Reserved
     BYTE13 : BYTE ;	// Reserved
     STR_MF1 : BOOL ;	// Modify M function number 1
     STR_MF2 : BOOL ;	// Modify M function number 2
     STR_MF3 : BOOL ;	// Modify M function number 3
     STR_MF4 : BOOL ;	// Modify M function number 4
     STR_MF5 : BOOL ;	// Modify M function number 5
     BIT14_5 : BOOL ;	// Reserved
     BIT14_6 : BOOL ;	// Reserved
     BIT14_7 : BOOL ;	// Reserved
     STR_TF1 : BOOL ;	// Modify T function number 1
     BIT15_1 : BOOL ;	// Reserved
     BIT15_2 : BOOL ;	// Reserved
     BIT15_3 : BOOL ;	// Reserved
     BIT15_4 : BOOL ;	// Reserved
     BIT15_5 : BOOL ;	// Reserved
     BIT15_6 : BOOL ;	// Reserved
     BIT15_7 : BOOL ;	// Reserved
     STR_HF1 : BOOL ;	// Modify H function number 1
     STR_HF2 : BOOL ;	// Modify H function number 2
     STR_HF3 : BOOL ;	// Modify H function number 3
     BIT16_3 : BOOL ;	// Reserved
     BIT16_4 : BOOL ;	// Reserved
     BIT16_5 : BOOL ;	// Reserved
     BIT16_6 : BOOL ;	// Reserved
     BIT16_7 : BOOL ;	// Reserved
     BYTE17 : BYTE ;	// Reserved
     NUM_M1 : BYTE ;	// M function number 1
     NUM_M2 : BYTE ;	// M function number 2
     NUM_M3 : BYTE ;	// M function number 3
     NUM_M4 : BYTE ;	// M function number 4
     NUM_M5 : BYTE ;	// M function number 5
     BYTE23 : BYTE ;	// Reserved
     NUM_T1 : WORD ;	// T function number 1
     NUM_H1 : WORD ;	// H function number 1
     FVAL_H1 : REAL ;	// H function value 1
     NUM_H2 : WORD ;	// H function number 2
     FVAL_H2 : REAL ;	// H function value 2
     NUM_H3 : WORD ;	// H function number 3
     FVAL_H3 : REAL ;	// H function value 3
     DWORD44 : DWORD ;	// Reserved
     WORD48 : WORD ;	// Reserved
     BYTE50_59 : ARRAY  [1 .. 10 ] OF BYTE ;	// Reserved
    END_STRUCT ;
   END_STRUCT ;
   WRJ1 : STRUCT 	// REQUEST 1 WRITE FM DATA
    BYTE0 : BYTE ;	// Reserved
    INP1 : BOOL ;	// Set digital ON-BOARD input 1
    INP2 : BOOL ;	// Set digital ON-BOARD input 2
    INP3 : BOOL ;	// Set digital ON-BOARD input 3
    INP4 : BOOL ;	// Set digital ON-BOARD input 4
    INP5 : BOOL ;	// Set digital ON-BOARD input 5
    INP6 : BOOL ;	// Set digital ON-BOARD input 6
    INP7 : BOOL ;	// Set digital ON-BOARD input 7
    INP8 : BOOL ;	// Set digital ON-BOARD input 8
    BYTE2 : BYTE ;	// Reserved
    INP9 : BOOL ;	// Set digital ON-BOARD input 9
    INP10 : BOOL ;	// Set digital ON-BOARD input 10
    INP11 : BOOL ;	// Set digital ON-BOARD input 11
    INP12 : BOOL ;	// Set digital ON-BOARD input 12
    BIT3_4 : BOOL ;	// Reserved
    BIT3_5 : BOOL ;	// Reserved
    BIT3_6 : BOOL ;	// Reserved
    BIT3_7 : BOOL ;	// Reserved
    DISA_INP1 : BOOL ;	// Disable digital ON-BOARD output 1
    DISA_INP2 : BOOL ;	// Disable digital ON-BOARD output 2
    DISA_INP3 : BOOL ;	// Disable digital ON-BOARD output 3
    DISA_INP4 : BOOL ;	// Disable digital ON-BOARD output 4
    DISA_INP5 : BOOL ;	// Disable digital ON-BOARD output 5
    DISA_INP6 : BOOL ;	// Disable digital ON-BOARD output 6
    DISA_INP7 : BOOL ;	// Disable digital ON-BOARD output 7
    DISA_INP8 : BOOL ;	// Disable digital ON-BOARD output 8
    BYTE5 : BYTE ;	// Reserved
    OUTP1 : BOOL ;	// Set digital ON-BOARD output 1
    OUTP2 : BOOL ;	// Set digital ON-BOARD output 2
    OUTP3 : BOOL ;	// Set digital ON-BOARD output 3
    OUTP4 : BOOL ;	// Set digital ON-BOARD output 4
    OUTP5 : BOOL ;	// Set digital ON-BOARD output 5
    OUTP6 : BOOL ;	// Set digital ON-BOARD output 6
    OUTP7 : BOOL ;	// Set digital ON-BOARD output 7
    OUTP8 : BOOL ;	// Set digital ON-BOARD output 8
    ST_OUTP1 : BOOL ;	// Input digital ON-BOARD output 1
    ST_OUTP2 : BOOL ;	// Input digital ON-BOARD output 2
    ST_OUTP3 : BOOL ;	// Input digital ON-BOARD output 3
    ST_OUTP4 : BOOL ;	// Input digital ON-BOARD output 4
    ST_OUTP5 : BOOL ;	// Input digital ON-BOARD output 5
    ST_OUTP6 : BOOL ;	// Input digital ON-BOARD output 6
    ST_OUTP7 : BOOL ;	// Input digital ON-BOARD output 7
    ST_OUTP8 : BOOL ;	// Input digital ON-BOARD output 8
    BYTE8 : BYTE ;	// Reserved
    EINP17 : BOOL ;	// Set digital input 17 (local P bus)
    EINP18 : BOOL ;	// Set digital input 18 (local P bus)
    EINP19 : BOOL ;	// Set digital input 19 (local P bus)
    EINP20 : BOOL ;	// Set digital input 20 (local P bus)
    EINP21 : BOOL ;	// Set digital input 21 (local P bus)
    EINP22 : BOOL ;	// Set digital input 22 (local P bus)
    EINP23 : BOOL ;	// Set digital input 23 (local P bus)
    EINP24 : BOOL ;	// Set digital input 24 (local P bus)
    BYTE10 : BYTE ;	// Reserved
    EINP25 : BOOL ;	// Set digital input 25 (local P bus)
    EINP26 : BOOL ;	// Set digital input 26 (local P bus)
    EINP27 : BOOL ;	// Set digital input 27 (local P bus)
    EINP28 : BOOL ;	// Set digital input 28 (local P bus)
    EINP29 : BOOL ;	// Set digital input 29 (local P bus)
    EINP30 : BOOL ;	// Set digital input 30 (local P bus)
    EINP31 : BOOL ;	// Set digital input 31 (local P bus)
    EINP32 : BOOL ;	// Set digital input 32 (local P bus)
    WORD12 : WORD ;	// Reserved
    WORD14 : WORD ;	// Reserved
    DISA_EOUTP9 : BOOL ;	// Disable digital output 9 (local P bus)
    DISA_EOUTP10 : BOOL ;	// Disable digital output 10 (local P bus)
    DISA_EOUTP11 : BOOL ;	// Disable digital output 11 (local P bus)
    DISA_EOUTP12 : BOOL ;	// Disable digital output 12 (local P bus)
    DISA_EOUTP13 : BOOL ;	// Disable digital output 13 (local P bus)
    DISA_EOUTP14 : BOOL ;	// Disable digital output 14 (local P bus)
    DISA_EOUTP15 : BOOL ;	// Disable digital output 15 (local P bus)
    DISA_EOUTP16 : BOOL ;	// Disable digital output 16 (local P bus)
    BYTE17 : BYTE ;	// Reserved
    EOUTP9 : BOOL ;	// Set digital output 9 (local P bus)
    EOUTP10 : BOOL ;	// Set digital output 10 (local P bus)
    EOUTP11 : BOOL ;	// Set digital output 11 (local P bus)
    EOUTP12 : BOOL ;	// Set digital output 12 (local P bus)
    EOUTP13 : BOOL ;	// Set digital output 13 (local P bus)
    EOUTP14 : BOOL ;	// Set digital output 14 (local P bus)
    EOUTP15 : BOOL ;	// Set digital output 15 (local P bus)
    EOUTP16 : BOOL ;	// Set digital output 16 (local P bus)
    ST_EOUTP9 : BOOL ;	// Input digital output 9 (local P bus)
    ST_EOUTP10 : BOOL ;	// Input digital output 10 (local P bus)
    ST_EOUTP11 : BOOL ;	// Input digital output 11 (local P bus)
    ST_EOUTP12 : BOOL ;	// Input digital output 12 (local P bus)
    ST_EOUTP13 : BOOL ;	// Input digital output 13 (local P bus)
    ST_EOUTP14 : BOOL ;	// Input digital output 14 (local P bus)
    ST_EOUTP15 : BOOL ;	// Input digital output 15 (local P bus)
    ST_EOUTP16 : BOOL ;	// Input digital output 16 (local P bus)
    DISA_EOUTP17 : BOOL ;	// Disable digital output 17 (local P bus)
    DISA_EOUTP18 : BOOL ;	// Disable digital output 18 (local P bus)
    DISA_EOUTP19 : BOOL ;	// Disable digital output 19 (local P bus)
    DISA_EOUTP20 : BOOL ;	// Disable digital output 20 (local P bus)
    DISA_EOUTP21 : BOOL ;	// Disable digital output 21 (local P bus)
    DISA_EOUTP22 : BOOL ;	// Disable digital output 22 (local P bus)
    DISA_EOUTP23 : BOOL ;	// Disable digital output 23 (local P bus)
    DISA_EOUTP24 : BOOL ;	// Disable digital output 24 (local P bus)
    BYTE21 : BYTE ;	// Reserved
    EOUTP17 : BOOL ;	// Set digital output 17 (local P bus)
    EOUTP18 : BOOL ;	// Set digital output 18 (local P bus)
    EOUTP19 : BOOL ;	// Set digital output 19 (local P bus)
    EOUTP20 : BOOL ;	// Set digital output 20 (local P bus)
    EOUTP21 : BOOL ;	// Set digital output 21 (local P bus)
    EOUTP22 : BOOL ;	// Set digital output 22 (local P bus)
    EOUTP23 : BOOL ;	// Set digital output 23 (local P bus)
    EOUTP24 : BOOL ;	// Set digital output 24 (local P bus)
    ST_EOUTP17 : BOOL ;	// Input digital output 17 (local P bus)
    ST_EOUTP18 : BOOL ;	// Input digital output 18 (local P bus)
    ST_EOUTP19 : BOOL ;	// Input digital output 19 (local P bus)
    ST_EOUTP20 : BOOL ;	// Input digital output 20 (local P bus)
    ST_EOUTP21 : BOOL ;	// Input digital output 21 (local P bus)
    ST_EOUTP22 : BOOL ;	// Input digital output 22 (local P bus)
    ST_EOUTP23 : BOOL ;	// Input digital output 23 (local P bus)
    ST_EOUTP24 : BOOL ;	// Input digital output 24 (local P bus)
    BYTE24_39 : ARRAY  [1 .. 16 ] OF BYTE ;	// Reserved
   END_STRUCT ;
   RDJ1 : STRUCT 	// REQUEST 1 READ FM DATA
    INP1 : BOOL ;	// Status digital ON-BOARD input 1
    INP2 : BOOL ;	// Status digital ON-BOARD input 2
    INP3 : BOOL ;	// Status digital ON-BOARD input 3
    INP4 : BOOL ;	// Status digital ON-BOARD input 4
    INP5 : BOOL ;	// Status digital ON-BOARD input 5
    INP6 : BOOL ;	// Status digital ON-BOARD input 6
    INP7 : BOOL ;	// Status digital ON-BOARD input 7
    INP8 : BOOL ;	// Status digital ON-BOARD input 8
    INP9 : BOOL ;	// Status digital ON-BOARD input 9
    INP10 : BOOL ;	// Status digital ON-BOARD input 10
    INP11 : BOOL ;	// Status digital ON-BOARD input 11
    INP12 : BOOL ;	// Status digital ON-BOARD input 12
    BIT1_4 : BOOL ;	// Reserved
    BIT1_5 : BOOL ;	// Reserved
    BIT1_6 : BOOL ;	// Reserved
    BIT1_7 : BOOL ;	// Reserved
    OUTP1 : BOOL ;	// Status digital ON-BOARD output 1
    OUTP2 : BOOL ;	// Status digital ON-BOARD output 2
    OUTP3 : BOOL ;	// Status digital ON-BOARD output 3
    OUTP4 : BOOL ;	// Status digital ON-BOARD output 4
    OUTP5 : BOOL ;	// Status digital ON-BOARD output 5
    OUTP6 : BOOL ;	// Status digital ON-BOARD output 6
    OUTP7 : BOOL ;	// Status digital ON-BOARD output 7
    OUTP8 : BOOL ;	// Status digital ON-BOARD output 8
    BYTE3 : BYTE ;	// Reserved
    EINP17 : BOOL ;	// Status digital input 17 (local P bus)
    EINP18 : BOOL ;	// Status digital input 18 (local P bus)
    EINP19 : BOOL ;	// Status digital input 19 (local P bus)
    EINP20 : BOOL ;	// Status digital input 20 (local P bus)
    EINP21 : BOOL ;	// Status digital input 21 (local P bus)
    EINP22 : BOOL ;	// Status digital input 22 (local P bus)
    EINP23 : BOOL ;	// Status digital input 23 (local P bus)
    EINP24 : BOOL ;	// Status digital input 24 (local P bus)
    EINP25 : BOOL ;	// Status digital input 25 (local P bus)
    EINP26 : BOOL ;	// Status digital input 26 (local P bus)
    EINP27 : BOOL ;	// Status digital input 27 (local P bus)
    EINP28 : BOOL ;	// Status digital input 28 (local P bus)
    EINP29 : BOOL ;	// Status digital input 29 (local P bus)
    EINP30 : BOOL ;	// Status digital input 30 (local P bus)
    EINP31 : BOOL ;	// Status digital input 31 (local P bus)
    EINP32 : BOOL ;	// Status digital input 32 (local P bus)
    WORD6 : WORD ;	// Reserved
    EOUTP9 : BOOL ;	// Status digital output 9  (local P bus)
    EOUTP10 : BOOL ;	// Status digital output 10 (local P bus)
    EOUTP11 : BOOL ;	// Status digital output 11 (local P bus)
    EOUTP12 : BOOL ;	// Status digital output 12 (local P bus)
    EOUTP13 : BOOL ;	// Status digital output 13 (local P bus)
    EOUTP14 : BOOL ;	// Status digital output 14 (local P bus)
    EOUTP15 : BOOL ;	// Status digital output 15 (local P bus)
    EOUTP16 : BOOL ;	// Status digital output 16 (local P bus)
    EOUTP17 : BOOL ;	// Status digital output 17 (local P bus)
    EOUTP18 : BOOL ;	// Status digital output 18 (local P bus)
    EOUTP19 : BOOL ;	// Status digital output 19 (local P bus)
    EOUTP20 : BOOL ;	// Status digital output 20 (local P bus)
    EOUTP21 : BOOL ;	// Status digital output 21 (local P bus)
    EOUTP22 : BOOL ;	// Status digital output 22 (local P bus)
    EOUTP23 : BOOL ;	// Status digital output 23 (local P bus)
    EOUTP24 : BOOL ;	// Status digital output 24 (local P bus)
    WORD10 : WORD ;	// Reserved
    BYTE12_39 : ARRAY  [1 .. 28 ] OF BYTE ;	// Reserved
   END_STRUCT ;
   WRJ2 : STRUCT 	// REQUEST 2 WRITE CHANNEL DATA
    CH : ARRAY  [1 .. 4 ] OF STRUCT
     DISA_SYN1 : BOOL ;	// Disable synchronized action ID 1
     DISA_SYN2 : BOOL ;	// Disable synchronized action ID 2
     DISA_SYN3 : BOOL ;	// Disable synchronized action ID 3
     DISA_SYN4 : BOOL ;	// Disable synchronized action ID 4
     DISA_SYN5 : BOOL ;	// Disable synchronized action ID 5
     DISA_SYN6 : BOOL ;	// Disable synchronized action ID 6
     DISA_SYN7 : BOOL ;	// Disable synchronized action ID 7
     DISA_SYN8 : BOOL ;	// Disable synchronized action ID 8
     BYTE1 : BYTE ;	// Reserved
     PRZONE_1 : BOOL ;	// Activate protection zone 1
     PRZONE_2 : BOOL ;	// Activate protection zone 2
     PRZONE_3 : BOOL ;	// Activate protection zone 3
     PRZONE_4 : BOOL ;	// Activate protection zone 4
     BIT2_4 : BOOL ;	// Reserved
     BIT2_5 : BOOL ;	// Reserved
     BIT2_6 : BOOL ;	// Reserved
     BIT2_7 : BOOL ;	// Reserved
     BYTE3 : BYTE ;	// Reserved
     BIT4_0 : BOOL ;	// Reserved
     BIT4_1 : BOOL ;	// Reserved
     BIT4_2 : BOOL ;	// Reserved
     BIT4_3 : BOOL ;	// Reserved
     PTP_TRAV : BOOL ;	// Point-to-point travel (FM357-H, 1st channel only)
     BIT4_5 : BOOL ;	// Reserved
     BIT4_6 : BOOL ;	// Reserved
     BIT4_7 : BOOL ;	// Reserved
     BYTE5 : BYTE ;	// Reserved
    END_STRUCT ;
    BYTE24_39 : ARRAY  [1 .. 15 ] OF BYTE ;	// Reserved
   END_STRUCT ;
   RDJ2 : STRUCT 	// REQUEST 2 READ CHANNEL DATA
    CH : ARRAY  [1 .. 4 ] OF STRUCT
     DISA_SYN1 : BOOL ;	// Synchronized action ID1 can be disabled by CPU
     DISA_SYN2 : BOOL ;	// Synchronized action ID2 can be disabled by CPU
     DISA_SYN3 : BOOL ;	// Synchronized action ID3 can be disabled by CPU
     DISA_SYN4 : BOOL ;	// Synchronized action ID4 can be disabled by CPU
     DISA_SYN5 : BOOL ;	// Synchronized action ID5 can be disabled by CPU
     DISA_SYN6 : BOOL ;	// Synchronized action ID6 can be disabled by CPU
     DISA_SYN7 : BOOL ;	// Synchronized action ID7 can be disabled by CPU
     DISA_SYN8 : BOOL ;	// Synchronized action ID8 can be disabled by CPU
     BYTE1 : BYTE ;	// Reserved
     PRZONE1 : BOOL ;	// Protection zone 1 pre-activated
     PRZONE2 : BOOL ;	// Protection zone 2 pre-activated
     PRZONE3 : BOOL ;	// Protection zone 3 pre-activated
     PRZONE4 : BOOL ;	// Protection zone 4 pre-activated
     BIT2_4 : BOOL ;	// Reserved
     BIT2_5 : BOOL ;	// Reserved
     BIT2_6 : BOOL ;	// Reserved
     BIT2_7 : BOOL ;	// Reserved
     BYTE3 : BYTE ;	// Reserved
     PRZONE1_VIOL : BOOL ;	// Protection zone 1 violated
     PRZONE2_VIOL : BOOL ;	// Protection zone 2 violated
     PRZONE3_VIOL : BOOL ;	// Protection zone 3 violated
     PRZONE4_VIOL : BOOL ;	// Protection zone 4 violated
     BIT4_4 : BOOL ;	// Reserved
     BIT4_5 : BOOL ;	// Reserved
     BIT4_6 : BOOL ;	// Reserved
     BIT4_7 : BOOL ;	// Reserved
     BYTE5 : BYTE ;	// Reserved
     BIT6_0 : BOOL ;	// Reserved
     BIT6_1 : BOOL ;	// Reserved
     BIT6_2 : BOOL ;	// Reserved
     BIT6_3 : BOOL ;	// Reserved
     BIT6_4 : BOOL ;	// Reserved
     BIT6_5 : BOOL ;	// Reserved
     PTP_TRAV : BOOL ;	// Point-to-point travel active (FM357-H 1st channel only)
     BIT6_7 : BOOL ;	// Reserved
     BIT7_0 : BOOL ;	// Reserved
     BIT7_1 : BOOL ;	// Reserved
     BIT7_2 : BOOL ;	// Reserved
     BIT7_3 : BOOL ;	// Reserved
     BIT7_4 : BOOL ;	// Reserved
     BIT7_5 : BOOL ;	// Reserved
     DRUN_FD : BOOL ;	// Dry run feed (FM357-H, 1st channel only)
     BIT7_7 : BOOL ;	// Reserved
    END_STRUCT ;
    DWORD32 : DWORD ;	// Reserved
    DWORD36 : DWORD ;	// Reserved
   END_STRUCT ;
   BYTE660_END : ARRAY  [1 .. 302 ] OF BYTE ;	// Reserved
  END_STRUCT ;	
BEGIN
END_DATA_BLOCK

DATA_BLOCK "DB_AXIES"	// DB 31
VERSION : 0.1
  STRUCT
   AX : ARRAY  [1 .. 5 ] OF STRUCT
    CTR : STRUCT 	// AXIS CONTROL SIGNALS
     OVERR : BYTE ;	// Override
     BIT1_0 : BOOL ;	// Reserved
     ACKN_FISTOP : BOOL ;	// Acknowledge Fixed Stop Reached
     SENS_FISTOP : BOOL ;	// Fixed stop sensor
     BIT1_3 : BOOL ;	// Reserved
     FOLLOWUP : BOOL ;	// Follow-up mode
     BIT1_5 : BOOL ;	// Reserved
     BIT1_6 : BOOL ;	// Reserved
     ACT_OVERR : BOOL ;	// Activate override
     SWCAM : BOOL ;	// Activate software cams
     CTR_EN : BOOL ;	// Controller enable
     DELDIS_TOGO : BOOL ;	// Axial delete distance to go
     CLAMP : BOOL ;	// Activate terminals
     BIT2_4 : BOOL ;	// Reserved
     BIT2_5 : BOOL ;	// Reserved
     BIT2_6 : BOOL ;	// Reserved
     BIT2_7 : BOOL ;	// Reserved
     BIT3_0 : BOOL ;	// Reserved
     FISTOP_EN : BOOL ;	// Enable travel to fixed stop
     BIT3_2 : BOOL ;	// Reserved
     BIT3_3 : BOOL ;	// Reserved
     BIT3_4 : BOOL ;	// Reserved
     BIT3_5 : BOOL ;	// Reserved
     BIT3_6 : BOOL ;	// Reserved
     BIT3_7 : BOOL ;	// Reserved
     BIT4_0 : BOOL ;	// Reserved
     BIT4_1 : BOOL ;	// Reserved
     BIT4_2 : BOOL ;	// Reserved
     FD_STOP : BOOL ;	// Feed STOP
     BIT4_4 : BOOL ;	// Reserved
     RTR_OVERL : BOOL ;	// Activate rapid traverse override
     DIR_M : BOOL ;	// MINUS direction
     DIR_P : BOOL ;	// PLUS direction
     BYTE5 : BYTE ;	// Reserved
     BYTE6 : BYTE ;	// Reserved
     HWLIMIT_M : BOOL ;	// Hardware limit switch MINUS
     HWLIMIT_P : BOOL ;	// Hardware limit switch PLUS
     SWLIMIT2_M : BOOL ;	// 2nd software limit switch MINUS
     SWLIMIT2_P : BOOL ;	// 2nd software limit switch PLUS
     BIT7_4 : BOOL ;	// Reserved
     BIT7_5 : BOOL ;	// Reserved
     BIT7_6 : BOOL ;	// Reserved
     REF_DELAY : BOOL ;	// Reference point approach delay
     ROT_MON : BOOL ;	// Stepper motor rotation monitor
     MODE_CONTROL : BOOL ;	// Axis control mode
     BIT8_2 : BOOL ;	// Reserved
     BIT8_3 : BOOL ;	// Reserved
     FOAX_OVERL : BOOL ;	// Enable following axis overlay
     BIT8_5 : BOOL ;	// Reserved
     BIT8_6 : BOOL ;	// Reserved
     BIT8_7 : BOOL ;	// Reserved
     BIT9_0 : BOOL ;	// Reserved
     BIT9_1 : BOOL ;	// Reserved
     BIT9_2 : BOOL ;	// Reserved
     BIT9_3 : BOOL ;	// Reserved
     BIT9_4 : BOOL ;	// Reserved
     OSSTOP_REVP : BOOL ;	// Oscillation, stop at next reversal point
     OSSTOP : BOOL ;	// Oscillation, stop
     BIT9_7 : BOOL ;	// Reserved
     BIT10_0 : BOOL ;	// Reserved
     BIT10_1 : BOOL ;	// Reserved
     BIT10_2 : BOOL ;	// Reserved
     BIT10_3 : BOOL ;	// Reserved
     START_GSYNRUN : BOOL ;	// Start gantry synchronism
     BIT10_5 : BOOL ;	// Reserved
     BIT10_6 : BOOL ;	// Reserved
     BIT10_7 : BOOL ;	// Reserved
     BYTE11 : BYTE ;	// Reserved
     BIT12_0 : BOOL ;	// Reserved
     RUP_ENC_QSTOP : BOOL ;	// Ramp-function generator rapid stop
     TORQ_LIM2 : BOOL ;	// Torque limit 2
     SPEED_SMOOTH : BOOL ;	// Speed setpoint smoothing
     BIT12_4 : BOOL ;	// Reserved
     BIT12_5 : BOOL ;	// Reserved
     BIT12_6 : BOOL ;	// Reserved
     BIT12_7 : BOOL ;	// Reserved
     PAR_A : BOOL ;	// Select parameter set A
     PAR_B : BOOL ;	// Select parameter set B
     PAR_C : BOOL ;	// Select parameter set C
     BIT13_3 : BOOL ;	// Reserved
     BIT13_4 : BOOL ;	// Reserved
     BIT13_5 : BOOL ;	// Reserved
     INTEGR_DISA : BOOL ;	// Integrator disable n controller
     PULSE_EN : BOOL ;	// Pulse enable
     DWORD14 : DWORD ;	// Reserved
     WORD18 : WORD ;	// Reserved
    END_STRUCT ;
    CHB : STRUCT 	// AXIS CHECKBACK SIGNALS
     BIT0_0 : BOOL ;	// Reserved
     BIT0_1 : BOOL ;	// Reserved
     BIT0_2 : BOOL ;	// Reserved
     BIT0_3 : BOOL ;	// Reserved
     REF_SYNC : BOOL ;	// Referenced, synchronized
     BIT0_5 : BOOL ;	// Reserved
     POSROD_C : BOOL ;	// Position reached (target range coarse)
     POSROD_F : BOOL ;	// Position reached (target range fine)
     BIT1_0 : BOOL ;	// Reserved
     BIT1_1 : BOOL ;	// Reserved
     BIT1_2 : BOOL ;	// Reserved
     FOLLOWUP : BOOL ;	// Follow-up mode active
     STAT : BOOL ;	// Axis stationary
     POSCTR : BOOL ;	// Position controller active
     SPEEDCTR : BOOL ;	// Speed controller active
     BIT1_7 : BOOL ;	// Reserved
     SWCAM : BOOL ;	// Software cams active
     BIT2_1 : BOOL ;	// Reserved
     BIT2_2 : BOOL ;	// Reserved
     MSR_EN : BOOL ;	// Measurement active
     TRAVFI_STOP : BOOL ;	// Travel to fixed stop active
     FI_STOP : BOOL ;	// Fixed stop reached
     BIT2_6 : BOOL ;	// Reserved
     BIT2_7 : BOOL ;	// Reserved
     MASTERAX : BOOL ;	// Masteraxis active
     FOAX : BOOL ;	// Following axis activ
     BIT3_2 : BOOL ;	// Reserved
     AX_ACCEL : BOOL ;	// Axis accelerating
     SYNC_RUN : BOOL ;	// Synchronization running
     BIT3_5 : BOOL ;	// Reserved
     GO_M : BOOL ;	// MINUS traverse
     GO_P : BOOL ;	// PLUS traverse
     INC1 : BOOL ;	// Increment size 1 increment
     INC10 : BOOL ;	// Increment size 10 increments
     INC100 : BOOL ;	// Increment size 100 increments
     INC1000 : BOOL ;	// Increment size 1000 increments
     INC10000 : BOOL ;	// Increment size 10000 increments
     INC_VAR : BOOL ;	// Increment variable (FM357-H)
     CONT_TRAV : BOOL ;	// Continuous traverse
     BIT4_7 : BOOL ;	// Reserved
     ATCHAN_A : BOOL ;	// Axis at channel A (binary)
     ATCHAN_B : BOOL ;	// Axis at channel B (binary)
     ATCHAN_C : BOOL ;	// Axis at channel C (binary)
     ATCHAN_D : BOOL ;	// Axis at channel D (binary)
     BIT5_4 : BOOL ;	// Reserved
     INTERCHANGE_P : BOOL ;	// Axis interchange possible
     NEUTRAL : BOOL ;	// Neutral status
     BIT5_7 : BOOL ;	// Reserved
     WORD6 : WORD ;	// Reserved
     SYNC_F : BOOL ;	// Synchronism fine
     SYNC_C : BOOL ;	// Synchronism coarse
     BIT8_2 : BOOL ;	// Reserved
     BIT8_3 : BOOL ;	// Reserved
     BLENDED_MOT : BOOL ;	// Blended motion activ
     SPEED_WARN : BOOL ;	// Threshold of speed warning reached
     ACCEL_WARN : BOOL ;	// Threshold of acceleration warning reached
     BIT8_7 : BOOL ;	// Reserved
     ERR_ROT_MON : BOOL ;	// Error in stepper motor rotation monitoring
     MODE_CONTROL : BOOL ;	// Axis control mode active
     BIT9_2 : BOOL ;	// Reserved
     BIT9_3 : BOOL ;	// Reserved
     BIT9_4 : BOOL ;	// Reserved
     BIT9_5 : BOOL ;	// Reserved
     OS_MOT : BOOL ;	// Oscillation motion active
     OS_ACT : BOOL ;	// Axis is oscillation axis
     BIT10_0 : BOOL ;	// Reserved
     BIT10_1 : BOOL ;	// Reserved
     GAN_TRLIM_EX : BOOL ;	// Gantry trip limit exceeded
     GAN_LIM_EX : BOOL ;	// Gantry warning limit exceeded
     GSYNRUN_RDY : BOOL ;	// Synchronism ready to start
     GANGR_SYN : BOOL ;	// Gantry grouping synchronized
     GAN_MASTAX : BOOL ;	// Gantry master axis
     GAN_AX : BOOL ;	// Gantry axis
     SETUP_MD : BOOL ;	// Setup mode
     RUP_ENC_DISA : BOOL ;	// Ramp generator disable
     TORQ_LIM2 : BOOL ;	// Torque limit 2
     SPEED_SMOOTH : BOOL ;	// Speed setpoint smoothing
     BIT11_4 : BOOL ;	// Reserved
     BIT11_5 : BOOL ;	// Reserved
     BIT11_6 : BOOL ;	// Reserved
     BIT11_7 : BOOL ;	// Reserved
     PAR_A : BOOL ;	// Active parameter set A
     PAR_B : BOOL ;	// Active parameter set B
     PAR_C : BOOL ;	// Active parameter set C
     BIT12_3 : BOOL ;	// Reserved
     BIT12_4 : BOOL ;	// Reserved
     DRV_RDY : BOOL ;	// Drive ready
     INTEGR_DISA : BOOL ;	// Integrator disable n controller
     PULSE_EN : BOOL ;	// Pulse enable
     TEMP_MOTOR : BOOL ;	// Motor temperature prewarning
     TEMP_HSINK : BOOL ;	// Heatsink temperature prewarning
     RAMP_COMPL : BOOL ;	// Ramp-up complete
     MD_MDX : BOOL ;	// |Md| < Mdx
     NACT_NMIN : BOOL ;	// |n act| < n min
     NACT_NX : BOOL ;	// |n act| < n x
     NACT_NSET : BOOL ;	// n act = n set
     MSG_FUNCT : BOOL ;	// Variable signalling function
     WORD14 : WORD ;	// Reserved
     DWORD16 : DWORD ;	// Reserved
     ACT_POS : REAL ;	// Actual value
     DIS_TOGO : REAL ;	// Distance to go
     WORD28 : WORD ;	// Reserved
    END_STRUCT ;
    CTRCA : STRUCT 	// CONTROL SIGNALS CPU AXIS
     BIT0_0 : BOOL ;	// Reserved
     BIT0_1 : BOOL ;	// Reserved
     BIT0_2 : BOOL ;	// Reserved
     BIT0_3 : BOOL ;	// Reserved
     BIT0_4 : BOOL ;	// Reserved
     BIT0_5 : BOOL ;	// Reserved
     BIT0_6 : BOOL ;	// Reserved
     CPUAX : BOOL ;	// Request CPU axis
     INCR : BOOL ;	// Traverse incremental
     DC : BOOL ;	// Traverse by shortest path
     INCH : BOOL ;	// Traverse in inches
     BIT2_3 : BOOL ;	// Reserved
     BIT2_4 : BOOL ;	// Reserved
     BIT2_5 : BOOL ;	// Reserved
     BIT2_6 : BOOL ;	// Reserved
     START : BOOL ;	// Start CPU axis
     POS : REAL ;	// Position of CPU axis
     FRATE : REAL ;	// Feedrate of CPU axis
     DWORD12 : DWORD ;	// Reserved
     BYTE15 : BYTE ;	// Reserved
     BIT16_0 : BOOL ;	// Reserved
     RESET_INDEPCPUAX : BOOL ;	// Reset independant CPU axis
     RESUME_INDEPCPUAX : BOOL ;	// Resume independant CPU axis
     BIT16_3 : BOOL ;	// Reserved
     BIT16_4 : BOOL ;	// Reserved
     BIT16_5 : BOOL ;	// Reserved
     STOP_INDEPCPUAX : BOOL ;	// Stop independant CPU axis
     INDEPCPUAX : BOOL ;	// Requirement: independant CPU axis
    END_STRUCT ;
    CHBCA : STRUCT 	// CHECKBACK SIGNALS CPU AXIS
     BIT0_0 : BOOL ;	// Reserved
     BIT0_1 : BOOL ;	// Reserved
     BIT0_2 : BOOL ;	// Reserved
     BIT0_3 : BOOL ;	// Reserved
     BIT0_4 : BOOL ;	// Reserved
     BIT0_5 : BOOL ;	// Reserved
     BIT0_6 : BOOL ;	// Reserved
     CPUAX : BOOL ;	// CPU axis
     BIT1_0 : BOOL ;	// Reserved
     ERR : BOOL ;	// Traversing error
     BIT1_2 : BOOL ;	// Reserved
     BIT1_3 : BOOL ;	// Reserved
     BIT1_4 : BOOL ;	// Reserved
     BIT1_5 : BOOL ;	// Reserved
     INPOS : BOOL ;	// Position reached
     ACTIV : BOOL ;	// CPU axis active
     ERR_NO : BYTE ;	// Error number for CPU axis
     RESET_INDEPCPUAX : BOOL ;	// Reset independant CPU axis
     INDEPCPUAX : BOOL ;	// Independant CPU axis
     ERR_INDEPCPUAX : BOOL ;	// Error independant CPU axis
     BIT3_3 : BOOL ;	// Reserved
     BIT3_4 : BOOL ;	// Reserved
     BIT3_5 : BOOL ;	// Reserved
     BIT3_6 : BOOL ;	// Reserved
     BIT3_7 : BOOL ;	// Reserved
    END_STRUCT ;
    RES : ARRAY  [1 .. 30 ] OF BYTE ;	// Reserved
   END_STRUCT ;
  END_STRUCT ;	
BEGIN
END_DATA_BLOCK

DATA_BLOCK DB 100
VERSION : 0.1
BEGIN
// 14 bytes; values not shown
END_DATA_BLOCK

DATA_BLOCK DB 105
VERSION : 0.0
BEGIN
// 148 bytes; values not shown
END_DATA_BLOCK

DATA_BLOCK DB 108
VERSION : 0.1
BEGIN
// 402 bytes; values not shown
END_DATA_BLOCK

DATA_BLOCK DB 110
VERSION : 0.1
BEGIN
// 4206 bytes; values not shown
END_DATA_BLOCK

DATA_BLOCK DB 115
AUTHOR : AuD_MCE8
FAMILY : FM357_2
NAME : USERDB
VERSION : 3.1
BEGIN
// 94 bytes; values not shown
END_DATA_BLOCK

DATA_BLOCK DB 121
AUTHOR : AuD_MCE8
FAMILY : FM357_2
NAME : VAR_ADDR
VERSION : 3.1
BEGIN
// 190 bytes; values not shown
END_DATA_BLOCK

DATA_BLOCK DB 141
AUTHOR : AuD_MCE8
FAMILY : FM357_2
VERSION : 0.0
FB 3
BEGIN
END_DATA_BLOCK

DATA_BLOCK DB 142
AUTHOR : AuD_MCE8
FAMILY : FM357_2
VERSION : 0.0
FB 3
BEGIN
END_DATA_BLOCK

DATA_BLOCK DB 143
AUTHOR : AuD_MCE8
FAMILY : FM357_2
VERSION : 0.0
FB 3
BEGIN
END_DATA_BLOCK

ORGANIZATION_BLOCK OB 1
VERSION : 1.0
BEGIN
// (block stored without names or comments; labels and parameter names are numbered)
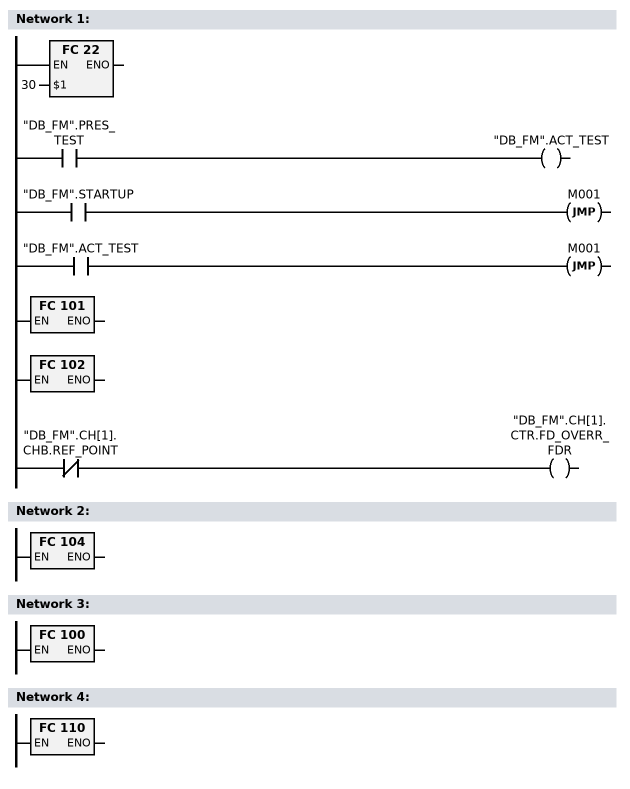
NETWORK
TITLE =
      CALL  FC 22 (
           $1                       := 30);
      A     "DB_FM".PRES_TEST;
      =     "DB_FM".ACT_TEST;
      A     "DB_FM".STARTUP;
      JC    M001;
      A     "DB_FM".ACT_TEST;
      JC    M001;
      CALL  FC 101;
      CALL  FC 102;
M001: NOP   0;
      AN    "DB_FM".CH[1].CHB.REF_POINT;
      =     "DB_FM".CH[1].CTR.FD_OVERR_FDR;
      NOP   0;
NETWORK
TITLE =
      CALL  FC 104;
      NOP   0;
NETWORK
TITLE =
      CALL  FC 100;
      NOP   0;
NETWORK
TITLE =
      CALL  FC 110;
      NOP   0;
END_ORGANIZATION_BLOCK

ORGANIZATION_BLOCK OB 82
VERSION : 1.0
BEGIN
// (block stored without names or comments; labels and parameter names are numbered)
NETWORK
TITLE =
      CALL  FC 5 (
           $1                       := 30);
      BE;
END_ORGANIZATION_BLOCK

ORGANIZATION_BLOCK OB 100
VERSION : 1.0
BEGIN
// (block stored without names or comments; labels and parameter names are numbered)
NETWORK
TITLE =
      CALL  FC 1 (
           $1                       := 30,
           $2                       := 300,
           $3                       := 100,
           $4                       := TRUE,
           $5                       := TRUE);
      BE;
END_ORGANIZATION_BLOCK

SYMBOL_TABLE
"READ_CLK"	SFC 1	SFC 1	// Read System Clock
"BLKMOV"	SFC 20	SFC 20	// Copy Variables
"CREAT_DB"	SFC 22	SFC 22	// Create Data Block
"DIS_AIRT"	SFC 41	SFC 41	// Delay the Higher Priority Interrupts and Asynchronous Errors
"EN_AIRT"	SFC 42	SFC 42	// Enable Higher Priority Interrupts and Asynchronous Errors
"STP"	SFC 46	SFC 46	// Change the CPU to STOP
"LGC_GADR"	SFC 49	SFC 49	// Query the Module Slot Belonging to a Logical Address
"RDSYSST"	SFC 51	SFC 51	// Read a System Status List or Partial List
"WR_USMSG"	SFC 52	SFC 52	// Write a User-Defined Diagnostic Event to the Diagnostic Buffer
"WR_REC"	SFC 58	SFC 58	// Write Data Record
"RD_REC"	SFC 59	SFC 59	// Read a Data Record
"CN"	UDT 1	UDT 1
"Axies"	UDT 2	UDT 2
"Udt_Axies"	UDT 4	UDT 4
"Udt_CN"	UDT 5	UDT 5
END_SYMBOL_TABLE

